   1:L PR[91] R[100]mm/sec CNT100;
   1:  PR[91,1] = PR[90,1] + -30.737;
   1:  PR[91,2] = PR[90,2] + -9.914;
   1:  PR[91,3] = PR[90,3] + 25.010;
   1:L PR[91] R[100]mm/sec CNT100;
   1:  PR[91,1] = PR[90,1] + -30.187;
   1:  PR[91,2] = PR[90,2] + -10.601;
   1:  PR[91,3] = PR[90,3] + 25.017;
   1:L PR[91] R[100]mm/sec CNT100;
   1:  PR[91,1] = PR[90,1] + -29.601;
   1:  PR[91,2] = PR[90,2] + -11.262;
   1:  PR[91,3] = PR[90,3] + 25.023;
   1:L PR[91] R[100]mm/sec CNT100;
   1:  PR[91,1] = PR[90,1] + -29.004;
   1:  PR[91,2] = PR[90,2] + -11.869;
   1:  PR[91,3] = PR[90,3] + 25.030;
   1:L PR[91] R[100]mm/sec CNT100;
   1:  PR[91,1] = PR[90,1] + -28.333;
   1:  PR[91,2] = PR[90,2] + -12.488;
   1:  PR[91,3] = PR[90,3] + 25.036;
   1:L PR[91] R[100]mm/sec CNT100;
   1:  PR[91,1] = PR[90,1] + -27.720;
   1:  PR[91,2] = PR[90,2] + -13.002;
   1:  PR[91,3] = PR[90,3] + 25.043;
   1:L PR[91] R[100]mm/sec CNT100;
   1:  PR[91,1] = PR[90,1] + -27.130;
   1:  PR[91,2] = PR[90,2] + -13.455;
   1:  PR[91,3] = PR[90,3] + 25.048;
   1:L PR[91] R[100]mm/sec CNT100;
   1:  PR[91,1] = PR[90,1] + -26.284;
   1:  PR[91,2] = PR[90,2] + -14.048;
   1:  PR[91,3] = PR[90,3] + 25.054;
   1:L PR[91] R[100]mm/sec CNT100;
   1:  PR[91,1] = PR[90,1] + -25.283;
   1:  PR[91,2] = PR[90,2] + -14.665;
   1:  PR[91,3] = PR[90,3] + 25.061;
   1:L PR[91] R[100]mm/sec CNT100;
   1:  PR[91,1] = PR[90,1] + -24.683;
   1:  PR[91,2] = PR[90,2] + -14.996;
   1:  PR[91,3] = PR[90,3] + 25.070;
   1:L PR[91] R[100]mm/sec CNT100;
   1:  PR[91,1] = PR[90,1] + -24.117;
   1:  PR[91,2] = PR[90,2] + -15.284;
   1:  PR[91,3] = PR[90,3] + 25.075;
   1:L PR[91] R[100]mm/sec CNT100;
   1:  PR[91,1] = PR[90,1] + -23.525;
   1:  PR[91,2] = PR[90,2] + -15.562;
   1:  PR[91,3] = PR[90,3] + 25.080;
   1:L PR[91] R[100]mm/sec CNT100;
   1:  PR[91,1] = PR[90,1] + -22.891;
   1:  PR[91,2] = PR[90,2] + -15.833;
   1:  PR[91,3] = PR[90,3] + 25.084;
   1:L PR[91] R[100]mm/sec CNT100;
   1:  PR[91,1] = PR[90,1] + -21.711;
   1:  PR[91,2] = PR[90,2] + -16.271;
   1:  PR[91,3] = PR[90,3] + 25.090;
   1:L PR[91] R[100]mm/sec CNT100;
   1:  PR[91,1] = PR[90,1] + -20.572;
   1:  PR[91,2] = PR[90,2] + -16.615;
   1:  PR[91,3] = PR[90,3] + 25.099;
   1:L PR[91] R[100]mm/sec CNT100;
   1:  PR[91,1] = PR[90,1] + -19.827;
   1:  PR[91,2] = PR[90,2] + -16.801;
   1:  PR[91,3] = PR[90,3] + 25.107;
   1:L PR[91] R[100]mm/sec CNT100;
   1:  PR[91,1] = PR[90,1] + -19.025;
   1:  PR[91,2] = PR[90,2] + -16.967;
   1:  PR[91,3] = PR[90,3] + 25.113;
   1:L PR[91] R[100]mm/sec CNT100;
   1:  PR[91,1] = PR[90,1] + -17.886;
   1:  PR[91,2] = PR[90,2] + -17.146;
   1:  PR[91,3] = PR[90,3] + 25.119;
   1:L PR[91] R[100]mm/sec CNT100;
   1:  PR[91,1] = PR[90,1] + -16.804;
   1:  PR[91,2] = PR[90,2] + -17.255;
   1:  PR[91,3] = PR[90,3] + 25.127;
   1:L PR[91] R[100]mm/sec CNT100;
   1:  PR[91,1] = PR[90,1] + -15.773;
   1:  PR[91,2] = PR[90,2] + -17.303;
   1:  PR[91,3] = PR[90,3] + 25.135;
   1:L PR[91] R[100]mm/sec CNT100;
   1:  PR[91,1] = PR[90,1] + -14.875;
   1:  PR[91,2] = PR[90,2] + -17.304;
   1:  PR[91,3] = PR[90,3] + 25.143;
   1:L PR[91] R[100]mm/sec CNT100;
   1:  PR[91,1] = PR[90,1] + -13.925;
   1:  PR[91,2] = PR[90,2] + -17.261;
   1:  PR[91,3] = PR[90,3] + 25.149;
   1:L PR[91] R[100]mm/sec CNT100;
   1:  PR[91,1] = PR[90,1] + -12.934;
   1:  PR[91,2] = PR[90,2] + -17.168;
   1:  PR[91,3] = PR[90,3] + 25.156;
   1:L PR[91] R[100]mm/sec CNT100;
   1:  PR[91,1] = PR[90,1] + -11.948;
   1:  PR[91,2] = PR[90,2] + -17.028;
   1:  PR[91,3] = PR[90,3] + 25.164;
   1:L PR[91] R[100]mm/sec CNT100;
   1:  PR[91,1] = PR[90,1] + -10.972;
   1:  PR[91,2] = PR[90,2] + -16.838;
   1:  PR[91,3] = PR[90,3] + 25.171;
   1:L PR[91] R[100]mm/sec CNT100;
   1:  PR[91,1] = PR[90,1] + -10.260;
   1:  PR[91,2] = PR[90,2] + -16.664;
   1:  PR[91,3] = PR[90,3] + 25.178;
   1:L PR[91] R[100]mm/sec CNT100;
   1:  PR[91,1] = PR[90,1] + -9.055;
   1:  PR[91,2] = PR[90,2] + -16.313;
   1:  PR[91,3] = PR[90,3] + 25.184;
   1:L PR[91] R[100]mm/sec CNT100;
   1:  PR[91,1] = PR[90,1] + -8.123;
   1:  PR[91,2] = PR[90,2] + -15.980;
   1:  PR[91,3] = PR[90,3] + 25.193;
   1:L PR[91] R[100]mm/sec CNT100;
   1:  PR[91,1] = PR[90,1] + -7.209;
   1:  PR[91,2] = PR[90,2] + -15.599;
   1:  PR[91,3] = PR[90,3] + 25.200;
   1:L PR[91] R[100]mm/sec CNT100;
   1:  PR[91,1] = PR[90,1] + -6.317;
   1:  PR[91,2] = PR[90,2] + -15.173;
   1:  PR[91,3] = PR[90,3] + 25.207;
   1:L PR[91] R[100]mm/sec CNT100;
   1:  PR[91,1] = PR[90,1] + -5.448;
   1:  PR[91,2] = PR[90,2] + -14.703;
   1:  PR[91,3] = PR[90,3] + 25.214;
   1:L PR[91] R[100]mm/sec CNT100;
   1:  PR[91,1] = PR[90,1] + -5.165;
   1:  PR[91,2] = PR[90,2] + -14.532;
   1:  PR[91,3] = PR[90,3] + 25.222;
   1:L PR[91] R[100]mm/sec CNT100;
   1:  PR[91,1] = PR[90,1] + -4.610;
   1:  PR[91,2] = PR[90,2] + -14.191;
   1:  PR[91,3] = PR[90,3] + 25.224;
   1:L PR[91] R[100]mm/sec CNT100;
   1:  PR[91,1] = PR[90,1] + -3.799;
   1:  PR[91,2] = PR[90,2] + -13.637;
   1:  PR[91,3] = PR[90,3] + 25.229;
   1:L PR[91] R[100]mm/sec CNT100;
   1:  PR[91,1] = PR[90,1] + -3.024;
   1:  PR[91,2] = PR[90,2] + -13.044;
   1:  PR[91,3] = PR[90,3] + 25.236;
   1:L PR[91] R[100]mm/sec CNT100;
   1:  PR[91,1] = PR[90,1] + -2.098;
   1:  PR[91,2] = PR[90,2] + -12.241;
   1:  PR[91,3] = PR[90,3] + 25.243;
   1:L PR[91] R[100]mm/sec CNT100;
   1:  PR[91,1] = PR[90,1] + -1.734;
   1:  PR[91,2] = PR[90,2] + -11.953;
   1:  PR[91,3] = PR[90,3] + 25.252;
   1:L PR[91] R[100]mm/sec CNT100;
   1:  PR[91,1] = PR[90,1] + -1.300;
   1:  PR[91,2] = PR[90,2] + -11.713;
   1:  PR[91,3] = PR[90,3] + 25.256;
   1:L PR[91] R[100]mm/sec CNT100;
   1:  PR[91,1] = PR[90,1] + -0.832;
   1:  PR[91,2] = PR[90,2] + -11.548;
   1:  PR[91,3] = PR[90,3] + 25.259;
   1:L PR[91] R[100]mm/sec CNT100;
   1:  PR[91,1] = PR[90,1] + -0.345;
   1:  PR[91,2] = PR[90,2] + -11.469;
   1:  PR[91,3] = PR[90,3] + 25.263;
   1:L PR[91] R[100]mm/sec CNT100;
   1:  PR[91,1] = PR[90,1] + 0.152;
   1:  PR[91,2] = PR[90,2] + -11.471;
   1:  PR[91,3] = PR[90,3] + 25.266;
   1:L PR[91] R[100]mm/sec CNT100;
   1:  PR[91] = PR[90];
   1:  PR[91,1] = PR[90,1] + 0.746;
   1:  PR[91,2] = PR[90,2] + -12.225;
   1:  PR[91,3] = PR[90,3] + 26.600;
   1:L PR[91] R[100]mm/sec CNT100;
   1:  PR[91,1] = PR[90,1] + 1.211;
   1:  PR[91,2] = PR[90,2] + -12.418;
   1:  PR[91,3] = PR[90,3] + 25.274;
   1:L PR[91] R[100]mm/sec CNT100;
   1:  PR[91,1] = PR[90,1] + 1.632;
   1:  PR[91,2] = PR[90,2] + -12.682;
   1:  PR[91,3] = PR[90,3] + 25.277;
   1:L PR[91] R[100]mm/sec CNT100;
   1:  PR[91,1] = PR[90,1] + 2.218;
   1:  PR[91,2] = PR[90,2] + -13.167;
   1:  PR[91,3] = PR[90,3] + 25.281;
   1:L PR[91] R[100]mm/sec CNT100;
   1:  PR[91,1] = PR[90,1] + 3.031;
   1:  PR[91,2] = PR[90,2] + -13.784;
   1:  PR[91,3] = PR[90,3] + 25.287;
   1:L PR[91] R[100]mm/sec CNT100;
   1:  PR[91,1] = PR[90,1] + 3.666;
   1:  PR[91,2] = PR[90,2] + -14.220;
   1:  PR[91,3] = PR[90,3] + 25.294;
   1:L PR[91] R[100]mm/sec CNT100;
   1:  PR[91,1] = PR[90,1] + 4.499;
   1:  PR[91,2] = PR[90,2] + -14.736;
   1:  PR[91,3] = PR[90,3] + 25.300;
   1:L PR[91] R[100]mm/sec CNT100;
   1:  PR[91,1] = PR[90,1] + 5.359;
   1:  PR[91,2] = PR[90,2] + -15.209;
   1:  PR[91,3] = PR[90,3] + 25.307;
   1:L PR[91] R[100]mm/sec CNT100;
   1:  PR[91,1] = PR[90,1] + 6.243;
   1:  PR[91,2] = PR[90,2] + -15.639;
   1:  PR[91,3] = PR[90,3] + 25.314;
   1:L PR[91] R[100]mm/sec CNT100;
   1:  PR[91,1] = PR[90,1] + 7.150;
   1:  PR[91,2] = PR[90,2] + -16.025;
   1:  PR[91,3] = PR[90,3] + 25.322;
   1:L PR[91] R[100]mm/sec CNT100;
   1:  PR[91,1] = PR[90,1] + 8.081;
   1:  PR[91,2] = PR[90,2] + -16.368;
   1:  PR[91,3] = PR[90,3] + 25.329;
   1:L PR[91] R[100]mm/sec CNT100;
   1:  PR[91,1] = PR[90,1] + 9.032;
   1:  PR[91,2] = PR[90,2] + -16.664;
   1:  PR[91,3] = PR[90,3] + 25.336;
   1:L PR[91] R[100]mm/sec CNT100;
   1:  PR[91,1] = PR[90,1] + 10.000;
   1:  PR[91,2] = PR[90,2] + -16.914;
   1:  PR[91,3] = PR[90,3] + 25.344;
   1:L PR[91] R[100]mm/sec CNT100;
   1:  PR[91,1] = PR[90,1] + 10.985;
   1:  PR[91,2] = PR[90,2] + -17.116;
   1:  PR[91,3] = PR[90,3] + 25.351;
   1:L PR[91] R[100]mm/sec CNT100;
   1:  PR[91,1] = PR[90,1] + 11.982;
   1:  PR[91,2] = PR[90,2] + -17.268;
   1:  PR[91,3] = PR[90,3] + 25.359;
   1:L PR[91] R[100]mm/sec CNT100;
   1:  PR[91,1] = PR[90,1] + 12.990;
   1:  PR[91,2] = PR[90,2] + -17.370;
   1:  PR[91,3] = PR[90,3] + 25.366;
   1:L PR[91] R[100]mm/sec CNT100;
   1:  PR[91,1] = PR[90,1] + 14.005;
   1:  PR[91,2] = PR[90,2] + -17.420;
   1:  PR[91,3] = PR[90,3] + 25.374;
   1:L PR[91] R[100]mm/sec CNT100;
   1:  PR[91,1] = PR[90,1] + 15.024;
   1:  PR[91,3] = PR[90,3] + 25.381;
   1:L PR[91] R[100]mm/sec CNT100;
   1:  PR[91,1] = PR[90,1] + 16.046;
   1:  PR[91,2] = PR[90,2] + -17.368;
   1:  PR[91,3] = PR[90,3] + 25.389;
   1:L PR[91] R[100]mm/sec CNT100;
   1:  PR[91,1] = PR[90,1] + 17.066;
   1:  PR[91,2] = PR[90,2] + -17.265;
   1:  PR[91,3] = PR[90,3] + 25.396;
   1:L PR[91] R[100]mm/sec CNT100;
   1:  PR[91,1] = PR[90,1] + 18.089;
   1:  PR[91,2] = PR[90,2] + -17.108;
   1:  PR[91,3] = PR[90,3] + 25.404;
   1:L PR[91] R[100]mm/sec CNT100;
   1:  PR[91,1] = PR[90,1] + 19.054;
   1:  PR[91,2] = PR[90,2] + -16.911;
   1:  PR[91,3] = PR[90,3] + 25.411;
   1:L PR[91] R[100]mm/sec CNT100;
   1:  PR[91,1] = PR[90,1] + 19.959;
   1:  PR[91,2] = PR[90,2] + -16.682;
   1:  PR[91,3] = PR[90,3] + 25.419;
   1:L PR[91] R[100]mm/sec CNT100;
   1:  PR[91,1] = PR[90,1] + 20.950;
   1:  PR[91,2] = PR[90,2] + -16.379;
   1:  PR[91,3] = PR[90,3] + 25.426;
   1:L PR[91] R[100]mm/sec CNT100;
   1:  PR[91,1] = PR[90,1] + 21.772;
   1:  PR[91,2] = PR[90,2] + -16.084;
   1:  PR[91,3] = PR[90,3] + 25.433;
   1:L PR[91] R[100]mm/sec CNT100;
   1:  PR[91,1] = PR[90,1] + 22.540;
   1:  PR[91,2] = PR[90,2] + -15.769;
   1:  PR[91,3] = PR[90,3] + 25.440;
   1:L PR[91] R[100]mm/sec CNT100;
   1:  PR[91,1] = PR[90,1] + 23.029;
   1:  PR[91,2] = PR[90,2] + -15.550;
   1:  PR[91,3] = PR[90,3] + 25.446;
   1:L PR[91] R[100]mm/sec CNT100;
   1:  PR[91,1] = PR[90,1] + 23.799;
   1:  PR[91,2] = PR[90,2] + -15.175;
   1:  PR[91,3] = PR[90,3] + 25.450;
   1:L PR[91] R[100]mm/sec CNT100;
   1:  PR[91,1] = PR[90,1] + 24.506;
   1:  PR[91,2] = PR[90,2] + -14.792;
   1:  PR[91,3] = PR[90,3] + 25.456;
   1:L PR[91] R[100]mm/sec CNT100;
   1:  PR[91,1] = PR[90,1] + 25.155;
   1:  PR[91,2] = PR[90,2] + -14.404;
   1:  PR[91,3] = PR[90,3] + 25.462;
   1:L PR[91] R[100]mm/sec CNT100;
   1:  PR[91,1] = PR[90,1] + 26.123;
   1:  PR[91,2] = PR[90,2] + -13.760;
   1:  PR[91,3] = PR[90,3] + 25.468;
   1:L PR[91] R[100]mm/sec CNT100;
   1:  PR[91,1] = PR[90,1] + 27.087;
   1:  PR[91,2] = PR[90,2] + -13.027;
   1:  PR[91,3] = PR[90,3] + 25.476;
   1:L PR[91] R[100]mm/sec CNT100;
   1:  PR[91,1] = PR[90,1] + 27.605;
   1:  PR[91,2] = PR[90,2] + -12.590;
   1:  PR[91,3] = PR[90,3] + 25.485;
   1:L PR[91] R[100]mm/sec CNT100;
   1:  PR[91,1] = PR[90,1] + 28.084;
   1:  PR[91,2] = PR[90,2] + -12.156;
   1:  PR[91,3] = PR[90,3] + 25.490;
   1:L PR[91] R[100]mm/sec CNT100;
   1:  PR[91,1] = PR[90,1] + 28.505;
   1:  PR[91,2] = PR[90,2] + -11.747;
   1:  PR[91,3] = PR[90,3] + 25.495;
   1:L PR[91] R[100]mm/sec CNT100;
   1:  PR[91,1] = PR[90,1] + 28.938;
   1:  PR[91,2] = PR[90,2] + -11.297;
   1:  PR[91,3] = PR[90,3] + 25.499;
   1:L PR[91] R[100]mm/sec CNT100;
   1:  PR[91,1] = PR[90,1] + 29.365;
   1:  PR[91,2] = PR[90,2] + -10.820;
   1:  PR[91,3] = PR[90,3] + 25.504;
   1:L PR[91] R[100]mm/sec CNT100;
   1:  PR[91,1] = PR[90,1] + 30.117;
   1:  PR[91,2] = PR[90,2] + -9.888;
   1:  PR[91,3] = PR[90,3] + 25.509;
   1:L PR[91] R[100]mm/sec CNT100;
   1:  PR[91,1] = PR[90,1] + 30.525;
   1:  PR[91,2] = PR[90,2] + -9.323;
   1:  PR[91,3] = PR[90,3] + 25.518;
   1:L PR[91] R[100]mm/sec CNT100;
   1:  PR[91,1] = PR[90,1] + 31.132;
   1:  PR[91,2] = PR[90,2] + -8.387;
   1:  PR[91,3] = PR[90,3] + 25.523;
   1:L PR[91] R[100]mm/sec CNT100;
   1:  PR[91,1] = PR[90,1] + 31.502;
   1:  PR[91,2] = PR[90,2] + -7.751;
   1:  PR[91,3] = PR[90,3] + 25.531;
   1:L PR[91] R[100]mm/sec CNT100;
   1:  PR[91,1] = PR[90,1] + 31.859;
   1:  PR[91,2] = PR[90,2] + -7.073;
   1:  PR[91,3] = PR[90,3] + 25.536;
   1:L PR[91] R[100]mm/sec CNT100;
   1:  PR[91,1] = PR[90,1] + 32.291;
   1:  PR[91,2] = PR[90,2] + -6.150;
   1:  PR[91,3] = PR[90,3] + 25.542;
   1:L PR[91] R[100]mm/sec CNT100;
   1:  PR[91,1] = PR[90,1] + 32.582;
   1:  PR[91,2] = PR[90,2] + -5.440;
   1:  PR[91,3] = PR[90,3] + 25.550;
   1:L PR[91] R[100]mm/sec CNT100;
   1:  PR[91,1] = PR[90,1] + 32.844;
   1:  PR[91,2] = PR[90,2] + -4.705;
   1:  PR[91,3] = PR[90,3] + 25.555;
   1:L PR[91] R[100]mm/sec CNT100;
   1:  PR[91,1] = PR[90,1] + 33.106;
   1:  PR[91,2] = PR[90,2] + -3.830;
   1:  PR[91,3] = PR[90,3] + 25.561;
   1:L PR[91] R[100]mm/sec CNT100;
   1:  PR[91,1] = PR[90,1] + 33.290;
   1:  PR[91,2] = PR[90,2] + -3.066;
   1:  PR[91,3] = PR[90,3] + 25.568;
   1:L PR[91] R[100]mm/sec CNT100;
   1:  PR[91,1] = PR[90,1] + 33.451;
   1:  PR[91,2] = PR[90,2] + -2.189;
   1:  PR[91,3] = PR[90,3] + 25.574;
   1:L PR[91] R[100]mm/sec CNT100;
   1:  PR[91,1] = PR[90,1] + 33.555;
   1:  PR[91,2] = PR[90,2] + -1.373;
   1:  PR[91,3] = PR[90,3] + 25.580;
   1:L PR[91] R[100]mm/sec CNT100;
   1:  PR[91,1] = PR[90,1] + 33.624;
   1:  PR[91,2] = PR[90,2] + -0.455;
   1:  PR[91,3] = PR[90,3] + 25.586;
   1:L PR[91] R[100]mm/sec CNT100;
   1:  PR[91,1] = PR[90,1] + 33.645;
   1:  PR[91,2] = PR[90,2] + 0.427;
   1:  PR[91,3] = PR[90,3] + 25.593;
   1:L PR[91] R[100]mm/sec CNT100;
   1:  PR[91,1] = PR[90,1] + 33.620;
   1:  PR[91,2] = PR[90,2] + 1.378;
   1:  PR[91,3] = PR[90,3] + 25.600;
   1:L PR[91] R[100]mm/sec CNT100;
   1:  PR[91,1] = PR[90,1] + 33.555;
   1:  PR[91,2] = PR[90,2] + 2.228;
   1:  PR[91,3] = PR[90,3] + 25.607;
   1:L PR[91] R[100]mm/sec CNT100;
   1:  PR[91,1] = PR[90,1] + 33.451;
   1:  PR[91,2] = PR[90,2] + 3.044;
   1:  PR[91,3] = PR[90,3] + 25.613;
   1:L PR[91] R[100]mm/sec CNT100;
   1:  PR[91,1] = PR[90,1] + 33.290;
   1:  PR[91,2] = PR[90,2] + 3.921;
   1:  PR[91,3] = PR[90,3] + 25.619;
   1:L PR[91] R[100]mm/sec CNT100;
   1:  PR[91,1] = PR[90,1] + 33.106;
   1:  PR[91,2] = PR[90,2] + 4.686;
   1:  PR[91,3] = PR[90,3] + 25.626;
   1:L PR[91] R[100]mm/sec CNT100;
   1:  PR[91,1] = PR[90,1] + 32.888;
   1:  PR[91,2] = PR[90,2] + 5.423;
   1:  PR[91,3] = PR[90,3] + 25.632;
   1:L PR[91] R[100]mm/sec CNT100;
   1:  PR[91,1] = PR[90,1] + 32.581;
   1:  PR[91,2] = PR[90,2] + 6.296;
   1:  PR[91,3] = PR[90,3] + 25.637;
   1:L PR[91] R[100]mm/sec CNT100;
   1:  PR[91,1] = PR[90,1] + 32.291;
   1:  PR[91,2] = PR[90,2] + 7.006;
   1:  PR[91,3] = PR[90,3] + 25.644;
   1:L PR[91] R[100]mm/sec CNT100;
   1:  PR[91,1] = PR[90,1] + 31.975;
   1:  PR[91,2] = PR[90,2] + 7.691;
   1:  PR[91,3] = PR[90,3] + 25.650;
   1:L PR[91] R[100]mm/sec CNT100;
   1:  PR[91,1] = PR[90,1] + 31.501;
   1:  PR[91,2] = PR[90,2] + 8.608;
   1:  PR[91,3] = PR[90,3] + 25.655;
   1:L PR[91] R[100]mm/sec CNT100;
   1:  PR[91,1] = PR[90,1] + 31.131;
   1:  PR[91,2] = PR[90,2] + 9.244;
   1:  PR[91,3] = PR[90,3] + 25.663;
   1:L PR[91] R[100]mm/sec CNT100;
   1:  PR[91,1] = PR[90,1] + 30.753;
   1:  PR[91,2] = PR[90,2] + 9.838;
   1:  PR[91,3] = PR[90,3] + 25.668;
   1:L PR[91] R[100]mm/sec CNT100;
   1:  PR[91,1] = PR[90,1] + 30.111;
   1:  PR[91,2] = PR[90,2] + 10.750;
   1:  PR[91,3] = PR[90,3] + 25.674;
   1:L PR[91] R[100]mm/sec CNT100;
   1:  PR[91,1] = PR[90,1] + 29.810;
   1:  PR[91,2] = PR[90,2] + 11.137;
   1:  PR[91,3] = PR[90,3] + 25.682;
   1:L PR[91] R[100]mm/sec CNT100;
   1:  PR[91,1] = PR[90,1] + 29.368;
   1:  PR[91,2] = PR[90,2] + 11.672;
   1:  PR[91,3] = PR[90,3] + 25.686;
   1:L PR[91] R[100]mm/sec CNT100;
   1:  PR[91,1] = PR[90,1] + 28.938;
   1:  PR[91,2] = PR[90,2] + 12.152;
   1:  PR[91,3] = PR[90,3] + 25.691;
   1:L PR[91] R[100]mm/sec CNT100;
   1:  PR[91,1] = PR[90,1] + 28.505;
   1:  PR[91,2] = PR[90,2] + 12.602;
   1:  PR[91,3] = PR[90,3] + 25.695;
   1:L PR[91] R[100]mm/sec CNT100;
   1:  PR[91,1] = PR[90,1] + 28.084;
   1:  PR[91,2] = PR[90,2] + 13.011;
   1:  PR[91,3] = PR[90,3] + 25.700;
   1:L PR[91] R[100]mm/sec CNT100;
   1:  PR[91,1] = PR[90,1] + 27.605;
   1:  PR[91,2] = PR[90,2] + 13.446;
   1:  PR[91,3] = PR[90,3] + 25.704;
   1:L PR[91] R[100]mm/sec CNT100;
   1:  PR[91,1] = PR[90,1] + 27.087;
   1:  PR[91,2] = PR[90,2] + 13.882;
   1:  PR[91,3] = PR[90,3] + 25.709;
   1:L PR[91] R[100]mm/sec CNT100;
   1:  PR[91,1] = PR[90,1] + 26.123;
   1:  PR[91,2] = PR[90,2] + 14.615;
   1:  PR[91,3] = PR[90,3] + 25.714;
   1:L PR[91] R[100]mm/sec CNT100;
   1:  PR[91,1] = PR[90,1] + 25.155;
   1:  PR[91,2] = PR[90,2] + 15.259;
   1:  PR[91,3] = PR[90,3] + 25.723;
   1:L PR[91] R[100]mm/sec CNT100;
   1:  PR[91,1] = PR[90,1] + 24.508;
   1:  PR[91,2] = PR[90,2] + 15.646;
   1:  PR[91,3] = PR[90,3] + 25.732;
   1:L PR[91] R[100]mm/sec CNT100;
   1:  PR[91,1] = PR[90,1] + 23.509;
   1:  PR[91,2] = PR[90,2] + 16.177;
   1:  PR[91,3] = PR[90,3] + 25.737;
   1:L PR[91] R[100]mm/sec CNT100;
   1:  PR[91,1] = PR[90,1] + 22.773;
   1:  PR[91,2] = PR[90,2] + 16.525;
   1:  PR[91,3] = PR[90,3] + 25.746;
   1:L PR[91] R[100]mm/sec CNT100;
   1:  PR[91,1] = PR[90,1] + 21.975;
   1:  PR[91,2] = PR[90,2] + 16.860;
   1:  PR[91,3] = PR[90,3] + 25.752;
   1:L PR[91] R[100]mm/sec CNT100;
   1:  PR[91,1] = PR[90,1] + 20.948;
   1:  PR[91,2] = PR[90,2] + 17.235;
   1:  PR[91,3] = PR[90,3] + 25.758;
   1:L PR[91] R[100]mm/sec CNT100;
   1:  PR[91,1] = PR[90,1] + 19.958;
   1:  PR[91,2] = PR[90,2] + 17.537;
   1:  PR[91,3] = PR[90,3] + 25.766;
   1:L PR[91] R[100]mm/sec CNT100;
   1:  PR[91,1] = PR[90,1] + 19.054;
   1:  PR[91,2] = PR[90,2] + 17.767;
   1:  PR[91,3] = PR[90,3] + 25.774;
   1:L PR[91] R[100]mm/sec CNT100;
   1:  PR[91,1] = PR[90,1] + 18.081;
   1:  PR[91,2] = PR[90,2] + 17.964;
   1:  PR[91,3] = PR[90,3] + 25.781;
   1:L PR[91] R[100]mm/sec CNT100;
   1:  PR[91,1] = PR[90,1] + 17.065;
   1:  PR[91,2] = PR[90,2] + 18.120;
   1:  PR[91,3] = PR[90,3] + 25.788;
   1:L PR[91] R[100]mm/sec CNT100;
   1:  PR[91,1] = PR[90,1] + 16.045;
   1:  PR[91,2] = PR[90,2] + 18.223;
   1:  PR[91,3] = PR[90,3] + 25.796;
   1:L PR[91] R[100]mm/sec CNT100;
   1:  PR[91,1] = PR[90,1] + 15.024;
   1:  PR[91,2] = PR[90,2] + 18.275;
   1:  PR[91,3] = PR[90,3] + 25.803;
   1:L PR[91] R[100]mm/sec CNT100;
   1:  PR[91,1] = PR[90,1] + 14.002;
   1:  PR[91,2] = PR[90,2] + 18.276;
   1:  PR[91,3] = PR[90,3] + 25.811;
   1:L PR[91] R[100]mm/sec CNT100;
   1:  PR[91,1] = PR[90,1] + 13.394;
   1:  PR[91,2] = PR[90,2] + 18.250;
   1:  PR[91,3] = PR[90,3] + 25.818;
   1:L PR[91] R[100]mm/sec CNT100;
   1:  PR[91,1] = PR[90,1] + 12.993;
   1:  PR[91,2] = PR[90,2] + 18.225;
   1:  PR[91,3] = PR[90,3] + 25.823;
   1:L PR[91] R[100]mm/sec CNT100;
   1:  PR[91,1] = PR[90,1] + 11.982;
   1:  PR[91,2] = PR[90,2] + 18.123;
   1:  PR[91,3] = PR[90,3] + 25.826;
   1:L PR[91] R[100]mm/sec CNT100;
   1:  PR[91,1] = PR[90,1] + 10.982;
   1:  PR[91,2] = PR[90,2] + 17.970;
   1:  PR[91,3] = PR[90,3] + 25.833;
   1:L PR[91] R[100]mm/sec CNT100;
   1:  PR[91,1] = PR[90,1] + 10.618;
   1:  PR[91,2] = PR[90,2] + 17.900;
   1:  PR[91,3] = PR[90,3] + 25.841;
   1:L PR[91] R[100]mm/sec CNT100;
   1:  PR[91,1] = PR[90,1] + 10.003;
   1:  PR[91,2] = PR[90,2] + 17.770;
   1:  PR[91,3] = PR[90,3] + 25.844;
   1:L PR[91] R[100]mm/sec CNT100;
   1:  PR[91,1] = PR[90,1] + 9.032;
   1:  PR[91,2] = PR[90,2] + 17.520;
   1:  PR[91,3] = PR[90,3] + 25.848;
   1:L PR[91] R[100]mm/sec CNT100;
   1:  PR[91,1] = PR[90,1] + 8.081;
   1:  PR[91,2] = PR[90,2] + 17.223;
   1:  PR[91,3] = PR[90,3] + 25.856;
   1:L PR[91] R[100]mm/sec CNT100;
   1:  PR[91,1] = PR[90,1] + 7.151;
   1:  PR[91,2] = PR[90,2] + 16.881;
   1:  PR[91,3] = PR[90,3] + 25.863;
   1:L PR[91] R[100]mm/sec CNT100;
   1:  PR[91,1] = PR[90,1] + 6.243;
   1:  PR[91,2] = PR[90,2] + 16.494;
   1:  PR[91,3] = PR[90,3] + 25.870;
   1:L PR[91] R[100]mm/sec CNT100;
   1:  PR[91,1] = PR[90,1] + 5.359;
   1:  PR[91,2] = PR[90,2] + 16.064;
   1:  PR[91,3] = PR[90,3] + 25.878;
   1:L PR[91] R[100]mm/sec CNT100;
   1:  PR[91,1] = PR[90,1] + 4.499;
   1:  PR[91,2] = PR[90,2] + 15.591;
   1:  PR[91,3] = PR[90,3] + 25.885;
   1:L PR[91] R[100]mm/sec CNT100;
   1:  PR[91,1] = PR[90,1] + 3.794;
   1:  PR[91,2] = PR[90,2] + 15.157;
   1:  PR[91,3] = PR[90,3] + 25.892;
   1:L PR[91] R[100]mm/sec CNT100;
   1:  PR[91,1] = PR[90,1] + 2.863;
   1:  PR[91,2] = PR[90,2] + 14.519;
   1:  PR[91,3] = PR[90,3] + 25.898;
   1:L PR[91] R[100]mm/sec CNT100;
   1:  PR[91,1] = PR[90,1] + 2.220;
   1:  PR[91,2] = PR[90,2] + 14.024;
   1:  PR[91,3] = PR[90,3] + 25.907;
   1:L PR[91] R[100]mm/sec CNT100;
   1:  PR[91,1] = PR[90,1] + 1.632;
   1:  PR[91,2] = PR[90,2] + 13.537;
   1:  PR[91,3] = PR[90,3] + 25.913;
   1:L PR[91] R[100]mm/sec CNT100;
   1:  PR[91,1] = PR[90,1] + 1.211;
   1:  PR[91,2] = PR[90,2] + 13.274;
   1:  PR[91,3] = PR[90,3] + 25.918;
   1:L PR[91] R[100]mm/sec CNT100;
   1:  PR[91,1] = PR[90,1] + 0.746;
   1:  PR[91,2] = PR[90,2] + 13.080;
   1:  PR[91,3] = PR[90,3] + 25.922;
   1:L PR[91] R[100]mm/sec CNT100;
   1:  PR[91,1] = PR[90,1] + 0.256;
   1:  PR[91,2] = PR[90,2] + 12.971;
   1:  PR[91,3] = PR[90,3] + 25.926;
   1:L PR[91] R[100]mm/sec CNT100;
   1:  PR[91,1] = PR[90,1] + -0.239;
   1:  PR[91,2] = PR[90,2] + 12.949;
   1:  PR[91,3] = PR[90,3] + 25.929;
   1:L PR[91] R[100]mm/sec CNT100;
   1:  PR[91,1] = PR[90,1] + -0.723;
   1:  PR[91,2] = PR[90,2] + 13.011;
   1:  PR[91,3] = PR[90,3] + 25.933;
   1:L PR[91] R[100]mm/sec CNT100;
   1:  PR[91,1] = PR[90,1] + -0.967;
   1:  PR[91,2] = PR[90,2] + 13.081;
   1:  PR[91,3] = PR[90,3] + 25.937;
   1:L PR[91] R[100]mm/sec CNT100;
   1:  PR[91,1] = PR[90,1] + -1.206;
   1:  PR[91,2] = PR[90,2] + 13.159;
   1:  PR[91,3] = PR[90,3] + 25.939;
   1:L PR[91] R[100]mm/sec CNT100;
   1:  PR[91,1] = PR[90,1] + -1.645;
   1:  PR[91,2] = PR[90,2] + 13.379;
   1:  PR[91,3] = PR[90,3] + 25.940;
   1:L PR[91] R[100]mm/sec CNT100;
   1:  PR[91,1] = PR[90,1] + -2.022;
   1:  PR[91,2] = PR[90,2] + 13.658;
   1:  PR[91,3] = PR[90,3] + 25.944;
   1:L PR[91] R[100]mm/sec CNT100;
   1:  PR[91,1] = PR[90,1] + -2.509;
   1:  PR[91,2] = PR[90,2] + 14.062;
   1:  PR[91,3] = PR[90,3] + 25.948;
   1:L PR[91] R[100]mm/sec CNT100;
   1:  PR[91,1] = PR[90,1] + -3.128;
   1:  PR[91,2] = PR[90,2] + 14.535;
   1:  PR[91,3] = PR[90,3] + 25.952;
   1:L PR[91] R[100]mm/sec CNT100;
   1:  PR[91,1] = PR[90,1] + -3.950;
   1:  PR[91,2] = PR[90,2] + 15.102;
   1:  PR[91,3] = PR[90,3] + 25.958;
   1:L PR[91] R[100]mm/sec CNT100;
   1:  PR[91,1] = PR[90,1] + -4.805;
   1:  PR[91,2] = PR[90,2] + 15.627;
   1:  PR[91,3] = PR[90,3] + 25.965;
   1:L PR[91] R[100]mm/sec CNT100;
   1:  PR[91,1] = PR[90,1] + -5.713;
   1:  PR[91,2] = PR[90,2] + 16.121;
   1:  PR[91,3] = PR[90,3] + 25.973;
   1:L PR[91] R[100]mm/sec CNT100;
   1:  PR[91,1] = PR[90,1] + -6.594;
   1:  PR[91,2] = PR[90,2] + 16.545;
   1:  PR[91,3] = PR[90,3] + 25.980;
   1:L PR[91] R[100]mm/sec CNT100;
   1:  PR[91,1] = PR[90,1] + -7.514;
   1:  PR[91,2] = PR[90,2] + 16.931;
   1:  PR[91,3] = PR[90,3] + 25.988;
   1:L PR[91] R[100]mm/sec CNT100;
   1:  PR[91,1] = PR[90,1] + -8.452;
   1:  PR[91,2] = PR[90,2] + 17.270;
   1:  PR[91,3] = PR[90,3] + 25.995;
   1:L PR[91] R[100]mm/sec CNT100;
   1:  PR[91,1] = PR[90,1] + -9.408;
   1:  PR[91,2] = PR[90,2] + 17.561;
   1:  PR[91,3] = PR[90,3] + 26.002;
   1:L PR[91] R[100]mm/sec CNT100;
   1:  PR[91,1] = PR[90,1] + -10.378;
   1:  PR[91,2] = PR[90,2] + 17.803;
   1:  PR[91,3] = PR[90,3] + 26.010;
   1:L PR[91] R[100]mm/sec CNT100;
   1:  PR[91,1] = PR[90,1] + -11.359;
   1:  PR[91,2] = PR[90,2] + 17.996;
   1:  PR[91,3] = PR[90,3] + 26.017;
   1:L PR[91] R[100]mm/sec CNT100;
   1:  PR[91,1] = PR[90,1] + -12.350;
   1:  PR[91,2] = PR[90,2] + 18.140;
   1:  PR[91,3] = PR[90,3] + 26.025;
   1:L PR[91] R[100]mm/sec CNT100;
   1:  PR[91,1] = PR[90,1] + -13.346;
   1:  PR[91,2] = PR[90,2] + 18.234;
   1:  PR[91,3] = PR[90,3] + 26.032;
   1:L PR[91] R[100]mm/sec CNT100;
   1:  PR[91,1] = PR[90,1] + -14.345;
   1:  PR[91,2] = PR[90,2] + 18.278;
   1:  PR[91,3] = PR[90,3] + 26.039;
   1:L PR[91] R[100]mm/sec CNT100;
   1:  PR[91,1] = PR[90,1] + -15.344;
   1:  PR[91,2] = PR[90,2] + 18.274;
   1:  PR[91,3] = PR[90,3] + 26.047;
   1:L PR[91] R[100]mm/sec CNT100;
   1:  PR[91,1] = PR[90,1] + -16.341;
   1:  PR[91,2] = PR[90,2] + 18.219;
   1:  PR[91,3] = PR[90,3] + 26.054;
   1:L PR[91] R[100]mm/sec CNT100;
   1:  PR[91,1] = PR[90,1] + -17.331;
   1:  PR[91,2] = PR[90,2] + 18.116;
   1:  PR[91,3] = PR[90,3] + 26.062;
   1:L PR[91] R[100]mm/sec CNT100;
   1:  PR[91,1] = PR[90,1] + -18.323;
   1:  PR[91,2] = PR[90,2] + 17.963;
   1:  PR[91,3] = PR[90,3] + 26.069;
   1:L PR[91] R[100]mm/sec CNT100;
   1:  PR[91,1] = PR[90,1] + -19.288;
   1:  PR[91,2] = PR[90,2] + 17.768;
   1:  PR[91,3] = PR[90,3] + 26.076;
   1:L PR[91] R[100]mm/sec CNT100;
   1:  PR[91,1] = PR[90,1] + -20.196;
   1:  PR[91,2] = PR[90,2] + 17.539;
   1:  PR[91,3] = PR[90,3] + 26.084;
   1:L PR[91] R[100]mm/sec CNT100;
   1:  PR[91,1] = PR[90,1] + -21.189;
   1:  PR[91,2] = PR[90,2] + 17.236;
   1:  PR[91,3] = PR[90,3] + 26.091;
   1:L PR[91] R[100]mm/sec CNT100;
   1:  PR[91,1] = PR[90,1] + -22.012;
   1:  PR[91,2] = PR[90,2] + 16.940;
   1:  PR[91,3] = PR[90,3] + 26.098;
   1:L PR[91] R[100]mm/sec CNT100;
   1:  PR[91,1] = PR[90,1] + -23.016;
   1:  PR[91,2] = PR[90,2] + 16.523;
   1:  PR[91,3] = PR[90,3] + 26.105;
   1:L PR[91] R[100]mm/sec CNT100;
   1:  PR[91,1] = PR[90,1] + -23.753;
   1:  PR[91,2] = PR[90,2] + 16.174;
   1:  PR[91,3] = PR[90,3] + 26.113;
   1:L PR[91] R[100]mm/sec CNT100;
   1:  PR[91,1] = PR[90,1] + -24.756;
   1:  PR[91,2] = PR[90,2] + 15.638;
   1:  PR[91,3] = PR[90,3] + 26.119;
   1:L PR[91] R[100]mm/sec CNT100;
   1:  PR[91,1] = PR[90,1] + -25.406;
   1:  PR[91,2] = PR[90,2] + 15.249;
   1:  PR[91,3] = PR[90,3] + 26.127;
   1:L PR[91] R[100]mm/sec CNT100;
   1:  PR[91,1] = PR[90,1] + -26.386;
   1:  PR[91,2] = PR[90,2] + 14.594;
   1:  PR[91,3] = PR[90,3] + 26.133;
   1:L PR[91] R[100]mm/sec CNT100;
   1:  PR[91,1] = PR[90,1] + -26.948;
   1:  PR[91,2] = PR[90,2] + 14.178;
   1:  PR[91,3] = PR[90,3] + 26.142;
   1:L PR[91] R[100]mm/sec CNT100;
   1:  PR[91,1] = PR[90,1] + -27.884;
   1:  PR[91,2] = PR[90,2] + 13.408;
   1:  PR[91,3] = PR[90,3] + 26.147;
   1:L PR[91] R[100]mm/sec CNT100;
   1:  PR[91,1] = PR[90,1] + -28.363;
   1:  PR[91,2] = PR[90,2] + 12.972;
   1:  PR[91,3] = PR[90,3] + 26.156;
   1:L PR[91] R[100]mm/sec CNT100;
   1:  PR[91,1] = PR[90,1] + -28.804;
   1:  PR[91,2] = PR[90,2] + 12.542;
   1:  PR[91,3] = PR[90,3] + 26.160;
   1:L PR[91] R[100]mm/sec CNT100;
   1:  PR[91,1] = PR[90,1] + -29.218;
   1:  PR[91,2] = PR[90,2] + 12.111;
   1:  PR[91,3] = PR[90,3] + 26.165;
   1:L PR[91] R[100]mm/sec CNT100;
   1:  PR[91,1] = PR[90,1] + -29.640;
   1:  PR[91,2] = PR[90,2] + 11.639;
   1:  PR[91,3] = PR[90,3] + 26.169;
   1:L PR[91] R[100]mm/sec CNT100;
   1:  PR[91,1] = PR[90,1] + -30.379;
   1:  PR[91,2] = PR[90,2] + 10.721;
   1:  PR[91,3] = PR[90,3] + 26.174;
   1:L PR[91] R[100]mm/sec CNT100;
   1:  PR[91,1] = PR[90,1] + -30.782;
   1:  PR[91,2] = PR[90,2] + 10.162;
   1:  PR[91,3] = PR[90,3] + 26.183;
   1:L PR[91] R[100]mm/sec CNT100;
   1:  PR[91,1] = PR[90,1] + -31.185;
   1:  PR[91,2] = PR[90,2] + 9.551;
   1:  PR[91,3] = PR[90,3] + 26.188;
   1:L PR[91] R[100]mm/sec CNT100;
   1:  PR[91,1] = PR[90,1] + -31.747;
   1:  PR[91,2] = PR[90,2] + 8.601;
   1:  PR[91,3] = PR[90,3] + 26.193;
   1:L PR[91] R[100]mm/sec CNT100;
   1:  PR[91,1] = PR[90,1] + -32.101;
   1:  PR[91,2] = PR[90,2] + 7.923;
   1:  PR[91,3] = PR[90,3] + 26.202;
   1:L PR[91] R[100]mm/sec CNT100;
   1:  PR[91,1] = PR[90,1] + -32.533;
   1:  PR[91,2] = PR[90,2] + 6.990;
   1:  PR[91,3] = PR[90,3] + 26.207;
   1:L PR[91] R[100]mm/sec CNT100;
   1:  PR[91,1] = PR[90,1] + -32.824;
   1:  PR[91,2] = PR[90,2] + 6.273;
   1:  PR[91,3] = PR[90,3] + 26.215;
   1:L PR[91] R[100]mm/sec CNT100;
   1:  PR[91,1] = PR[90,1] + -33.086;
   1:  PR[91,2] = PR[90,2] + 5.533;
   1:  PR[91,3] = PR[90,3] + 26.221;
   1:L PR[91] R[100]mm/sec CNT100;
   1:  PR[91,1] = PR[90,1] + -33.315;
   1:  PR[91,2] = PR[90,2] + 4.772;
   1:  PR[91,3] = PR[90,3] + 26.226;
   1:L PR[91] R[100]mm/sec CNT100;
   1:  PR[91,1] = PR[90,1] + -33.531;
   1:  PR[91,2] = PR[90,2] + 3.892;
   1:  PR[91,3] = PR[90,3] + 26.232;
   1:L PR[91] R[100]mm/sec CNT100;
   1:  PR[91,1] = PR[90,1] + -33.691;
   1:  PR[91,2] = PR[90,2] + 3.023;
   1:  PR[91,3] = PR[90,3] + 26.239;
   1:L PR[91] R[100]mm/sec CNT100;
   1:  PR[91,1] = PR[90,1] + -33.795;
   1:  PR[91,2] = PR[90,2] + 2.215;
   1:  PR[91,3] = PR[90,3] + 26.245;
   1:L PR[91] R[100]mm/sec CNT100;
   1:  PR[91,1] = PR[90,1] + -33.859;
   1:  PR[91,2] = PR[90,2] + 1.371;
   1:  PR[91,3] = PR[90,3] + 26.251;
   1:L PR[91] R[100]mm/sec CNT100;
   1:  PR[91,1] = PR[90,1] + -33.883;
   1:  PR[91,2] = PR[90,2] + 0.428;
   1:  PR[91,3] = PR[90,3] + 26.258;
   1:L PR[91] R[100]mm/sec CNT100;
   1:  PR[91,1] = PR[90,1] + -33.859;
   1:  PR[91,2] = PR[90,2] + -0.516;
   1:  PR[91,3] = PR[90,3] + 26.265;
   1:L PR[91] R[100]mm/sec CNT100;
   1:  PR[91,1] = PR[90,1] + -33.795;
   1:  PR[91,2] = PR[90,2] + -1.359;
   1:  PR[91,3] = PR[90,3] + 26.272;
   1:L PR[91] R[100]mm/sec CNT100;
   1:  PR[91,1] = PR[90,1] + -33.678;
   1:  PR[91,2] = PR[90,2] + -2.249;
   1:  PR[91,3] = PR[90,3] + 26.278;
   1:L PR[91] R[100]mm/sec CNT100;
   1:  PR[91,1] = PR[90,1] + -33.550;
   1:  PR[91,2] = PR[90,2] + -2.942;
   1:  PR[91,3] = PR[90,3] + 26.285;
   1:L PR[91] R[100]mm/sec CNT100;
   1:  PR[91,1] = PR[90,1] + -33.314;
   1:  PR[91,2] = PR[90,2] + -3.918;
   1:  PR[91,3] = PR[90,3] + 26.290;
   1:L PR[91] R[100]mm/sec CNT100;
   1:  PR[91,1] = PR[90,1] + -33.086;
   1:  PR[91,2] = PR[90,2] + -4.678;
   1:  PR[91,3] = PR[90,3] + 26.297;
   1:L PR[91] R[100]mm/sec CNT100;
   1:  PR[91,1] = PR[90,1] + -32.825;
   1:  PR[91,2] = PR[90,2] + -5.416;
   1:  PR[91,3] = PR[90,3] + 26.303;
   1:L PR[91] R[100]mm/sec CNT100;
   1:  PR[91,1] = PR[90,1] + -32.440;
   1:  PR[91,2] = PR[90,2] + -6.346;
   1:  PR[91,3] = PR[90,3] + 26.309;
   1:L PR[91] R[100]mm/sec CNT100;
   1:  PR[91,1] = PR[90,1] + -32.102;
   1:  PR[91,2] = PR[90,2] + -7.066;
   1:  PR[91,3] = PR[90,3] + 26.316;
   1:L PR[91] R[100]mm/sec CNT100;
   1:  PR[91,1] = PR[90,1] + -31.747;
   1:  PR[91,2] = PR[90,2] + -7.745;
   1:  PR[91,3] = PR[90,3] + 26.322;
   1:L PR[91] R[100]mm/sec CNT100;
   1:  PR[91,1] = PR[90,1] + -31.185;
   1:  PR[91,2] = PR[90,2] + -8.695;
   1:  PR[91,3] = PR[90,3] + 26.328;
   1:L PR[91] R[100]mm/sec CNT100;
   1:  PR[91,1] = PR[90,1] + -30.782;
   1:  PR[91,2] = PR[90,2] + -9.307;
   1:  PR[91,3] = PR[90,3] + 26.336;
   1:L PR[91] R[100]mm/sec CNT100;
   1:  PR[91,1] = PR[90,1] + -30.379;
   1:  PR[91,2] = PR[90,2] + -9.866;
   1:  PR[91,3] = PR[90,3] + 26.341;
   1:L PR[91] R[100]mm/sec CNT100;
   1:  PR[91,1] = PR[90,1] + -29.640;
   1:  PR[91,2] = PR[90,2] + -10.784;
   1:  PR[91,3] = PR[90,3] + 26.347;
   1:L PR[91] R[100]mm/sec CNT100;
   1:  PR[91,1] = PR[90,1] + -29.218;
   1:  PR[91,2] = PR[90,2] + -11.256;
   1:  PR[91,3] = PR[90,3] + 26.355;
   1:L PR[91] R[100]mm/sec CNT100;
   1:  PR[91,1] = PR[90,1] + -28.788;
   1:  PR[91,2] = PR[90,2] + -11.704;
   1:  PR[91,3] = PR[90,3] + 26.360;
   1:L PR[91] R[100]mm/sec CNT100;
   1:  PR[91,1] = PR[90,1] + -28.363;
   1:  PR[91,2] = PR[90,2] + -12.117;
   1:  PR[91,3] = PR[90,3] + 26.365;
   1:L PR[91] R[100]mm/sec CNT100;
   1:  PR[91,1] = PR[90,1] + -27.884;
   1:  PR[91,2] = PR[90,2] + -12.553;
   1:  PR[91,3] = PR[90,3] + 26.369;
   1:L PR[91] R[100]mm/sec CNT100;
   1:  PR[91,1] = PR[90,1] + -26.948;
   1:  PR[91,2] = PR[90,2] + -13.322;
   1:  PR[91,3] = PR[90,3] + 26.374;
   1:L PR[91] R[100]mm/sec CNT100;
   1:  PR[91,1] = PR[90,1] + -26.383;
   1:  PR[91,2] = PR[90,2] + -13.741;
   1:  PR[91,3] = PR[90,3] + 26.383;
   1:L PR[91] R[100]mm/sec CNT100;
   1:  PR[91,1] = PR[90,1] + -25.769;
   1:  PR[91,2] = PR[90,2] + -14.160;
   1:  PR[91,3] = PR[90,3] + 26.388;
   1:L PR[91] R[100]mm/sec CNT100;
   1:  PR[91,1] = PR[90,1] + -24.753;
   1:  PR[91,2] = PR[90,2] + -14.785;
   1:  PR[91,3] = PR[90,3] + 26.393;
   1:L PR[91] R[100]mm/sec CNT100;
   1:  PR[91,1] = PR[90,1] + -23.755;
   1:  PR[91,2] = PR[90,2] + -15.318;
   1:  PR[91,3] = PR[90,3] + 26.402;
   1:L PR[91] R[100]mm/sec CNT100;
   1:  PR[91,1] = PR[90,1] + -22.778;
   1:  PR[91,2] = PR[90,2] + -15.770;
   1:  PR[91,3] = PR[90,3] + 26.411;
   1:L PR[91] R[100]mm/sec CNT100;
   1:  PR[91,1] = PR[90,1] + -22.013;
   1:  PR[91,2] = PR[90,2] + -16.085;
   1:  PR[91,3] = PR[90,3] + 26.419;
   1:L PR[91] R[100]mm/sec CNT100;
   1:  PR[91,1] = PR[90,1] + -21.189;
   1:  PR[91,2] = PR[90,2] + -16.381;
   1:  PR[91,3] = PR[90,3] + 26.425;
   1:L PR[91] R[100]mm/sec CNT100;
   1:  PR[91,1] = PR[90,1] + -20.300;
   1:  PR[91,2] = PR[90,2] + -16.655;
   1:  PR[91,3] = PR[90,3] + 26.431;
   1:L PR[91] R[100]mm/sec CNT100;
   1:  PR[91,1] = PR[90,1] + -19.288;
   1:  PR[91,2] = PR[90,2] + -16.913;
   1:  PR[91,3] = PR[90,3] + 26.438;
   1:L PR[91] R[100]mm/sec CNT100;
   1:  PR[91,1] = PR[90,1] + -18.316;
   1:  PR[91,2] = PR[90,2] + -17.110;
   1:  PR[91,3] = PR[90,3] + 26.446;
   1:L PR[91] R[100]mm/sec CNT100;
   1:  PR[91,1] = PR[90,1] + -17.332;
   1:  PR[91,2] = PR[90,2] + -17.261;
   1:  PR[91,3] = PR[90,3] + 26.453;
   1:L PR[91] R[100]mm/sec CNT100;
   1:  PR[91,1] = PR[90,1] + -16.341;
   1:  PR[91,2] = PR[90,2] + -17.364;
   1:  PR[91,3] = PR[90,3] + 26.460;
   1:L PR[91] R[100]mm/sec CNT100;
   1:  PR[91,1] = PR[90,1] + -15.344;
   1:  PR[91,2] = PR[90,2] + -17.418;
   1:  PR[91,3] = PR[90,3] + 26.468;
   1:L PR[91] R[100]mm/sec CNT100;
   1:  PR[91,1] = PR[90,1] + -14.345;
   1:  PR[91,2] = PR[90,2] + -17.423;
   1:  PR[91,3] = PR[90,3] + 26.475;
   1:L PR[91] R[100]mm/sec CNT100;
   1:  PR[91,1] = PR[90,1] + -13.345;
   1:  PR[91,2] = PR[90,2] + -17.379;
   1:  PR[91,3] = PR[90,3] + 26.483;
   1:L PR[91] R[100]mm/sec CNT100;
   1:  PR[91,1] = PR[90,1] + -12.822;
   1:  PR[91,2] = PR[90,2] + -17.331;
   1:  PR[91,3] = PR[90,3] + 26.490;
   1:L PR[91] R[100]mm/sec CNT100;
   1:  PR[91,1] = PR[90,1] + -12.351;
   1:  PR[91,2] = PR[90,2] + -17.285;
   1:  PR[91,3] = PR[90,3] + 26.494;
   1:L PR[91] R[100]mm/sec CNT100;
   1:  PR[91,1] = PR[90,1] + -11.359;
   1:  PR[91,2] = PR[90,2] + -17.141;
   1:  PR[91,3] = PR[90,3] + 26.497;
   1:L PR[91] R[100]mm/sec CNT100;
   1:  PR[91,1] = PR[90,1] + -10.378;
   1:  PR[91,2] = PR[90,2] + -16.948;
   1:  PR[91,3] = PR[90,3] + 26.505;
   1:L PR[91] R[100]mm/sec CNT100;
   1:  PR[91,1] = PR[90,1] + -9.410;
   1:  PR[91,2] = PR[90,2] + -16.706;
   1:  PR[91,3] = PR[90,3] + 26.512;
   1:L PR[91] R[100]mm/sec CNT100;
   1:  PR[91,1] = PR[90,1] + -8.290;
   1:  PR[91,2] = PR[90,2] + -16.357;
   1:  PR[91,3] = PR[90,3] + 26.520;
   1:L PR[91] R[100]mm/sec CNT100;
   1:  PR[91,1] = PR[90,1] + -7.514;
   1:  PR[91,2] = PR[90,2] + -16.076;
   1:  PR[91,3] = PR[90,3] + 26.528;
   1:L PR[91] R[100]mm/sec CNT100;
   1:  PR[91,1] = PR[90,1] + -6.594;
   1:  PR[91,2] = PR[90,2] + -15.689;
   1:  PR[91,3] = PR[90,3] + 26.534;
   1:L PR[91] R[100]mm/sec CNT100;
   1:  PR[91,1] = PR[90,1] + -5.691;
   1:  PR[91,2] = PR[90,2] + -15.255;
   1:  PR[91,3] = PR[90,3] + 26.542;
   1:L PR[91] R[100]mm/sec CNT100;
   1:  PR[91,1] = PR[90,1] + -4.804;
   1:  PR[91,2] = PR[90,2] + -14.772;
   1:  PR[91,3] = PR[90,3] + 26.549;
   1:L PR[91] R[100]mm/sec CNT100;
   1:  PR[91,1] = PR[90,1] + -3.950;
   1:  PR[91,2] = PR[90,2] + -14.247;
   1:  PR[91,3] = PR[90,3] + 26.557;
   1:L PR[91] R[100]mm/sec CNT100;
   1:  PR[91,1] = PR[90,1] + -3.128;
   1:  PR[91,2] = PR[90,2] + -13.680;
   1:  PR[91,3] = PR[90,3] + 26.564;
   1:L PR[91] R[100]mm/sec CNT100;
   1:  PR[91,1] = PR[90,1] + -2.487;
   1:  PR[91,2] = PR[90,2] + -13.189;
   1:  PR[91,3] = PR[90,3] + 26.571;
   1:L PR[91] R[100]mm/sec CNT100;
   1:  PR[91,1] = PR[90,1] + -2.021;
   1:  PR[91,2] = PR[90,2] + -12.801;
   1:  PR[91,3] = PR[90,3] + 26.577;
   1:L PR[91] R[100]mm/sec CNT100;
   1:  PR[91,1] = PR[90,1] + -1.644;
   1:  PR[91,2] = PR[90,2] + -12.523;
   1:  PR[91,3] = PR[90,3] + 26.582;
   1:L PR[91] R[100]mm/sec CNT100;
   1:  PR[91,1] = PR[90,1] + -1.206;
   1:  PR[91,2] = PR[90,2] + -12.304;
   1:  PR[91,3] = PR[90,3] + 26.585;
   1:L PR[91] R[100]mm/sec CNT100;
   1:  PR[91,1] = PR[90,1] + -0.967;
   1:  PR[91,2] = PR[90,2] + -12.225;
   1:  PR[91,3] = PR[90,3] + 26.589;
   1:L PR[91] R[100]mm/sec CNT100;
   1:  PR[91,1] = PR[90,1] + -0.723;
   1:  PR[91,2] = PR[90,2] + -12.155;
   1:  PR[91,3] = PR[90,3] + 26.591;
   1:L PR[91] R[100]mm/sec CNT100;
   1:  PR[91,1] = PR[90,1] + -0.239;
   1:  PR[91,2] = PR[90,2] + -12.094;
   1:  PR[91,3] = PR[90,3] + 26.593;
   1:L PR[91] R[100]mm/sec CNT100;
   1:  PR[91,1] = PR[90,1] + 0.256;
   1:  PR[91,2] = PR[90,2] + -12.116;
   1:  PR[91,3] = PR[90,3] + 26.596;
   1:L PR[91] R[100]mm/sec CNT100;
   1:  PR[91] = PR[90];
   1:  PR[91,1] = PR[90,1] + 0.840;
   1:  PR[91,2] = PR[90,2] + -12.856;
   1:  PR[91,3] = PR[90,3] + 27.930;
   1:L PR[91] R[100]mm/sec CNT100;
   1:  PR[91,1] = PR[90,1] + 1.300;
   1:  PR[91,2] = PR[90,2] + -13.063;
   1:  PR[91,3] = PR[90,3] + 26.604;
   1:L PR[91] R[100]mm/sec CNT100;
   1:  PR[91,1] = PR[90,1] + 1.701;
   1:  PR[91,2] = PR[90,2] + -13.334;
   1:  PR[91,3] = PR[90,3] + 26.608;
   1:L PR[91] R[100]mm/sec CNT100;
   1:  PR[91,1] = PR[90,1] + 2.162;
   1:  PR[91,2] = PR[90,2] + -13.692;
   1:  PR[91,3] = PR[90,3] + 26.611;
   1:L PR[91] R[100]mm/sec CNT100;
   1:  PR[91,1] = PR[90,1] + 2.968;
   1:  PR[91,2] = PR[90,2] + -14.260;
   1:  PR[91,3] = PR[90,3] + 26.615;
   1:L PR[91] R[100]mm/sec CNT100;
   1:  PR[91,1] = PR[90,1] + 3.805;
   1:  PR[91,2] = PR[90,2] + -14.788;
   1:  PR[91,3] = PR[90,3] + 26.623;
   1:L PR[91] R[100]mm/sec CNT100;
   1:  PR[91,1] = PR[90,1] + 4.259;
   1:  PR[91,2] = PR[90,2] + -15.046;
   1:  PR[91,3] = PR[90,3] + 26.630;
   1:L PR[91] R[100]mm/sec CNT100;
   1:  PR[91,1] = PR[90,1] + 4.664;
   1:  PR[91,2] = PR[90,2] + -15.268;
   1:  PR[91,3] = PR[90,3] + 26.634;
   1:L PR[91] R[100]mm/sec CNT100;
   1:  PR[91,1] = PR[90,1] + 5.555;
   1:  PR[91,2] = PR[90,2] + -15.708;
   1:  PR[91,3] = PR[90,3] + 26.638;
   1:L PR[91] R[100]mm/sec CNT100;
   1:  PR[91,1] = PR[90,1] + 6.467;
   1:  PR[91,2] = PR[90,2] + -16.102;
   1:  PR[91,3] = PR[90,3] + 26.645;
   1:L PR[91] R[100]mm/sec CNT100;
   1:  PR[91,1] = PR[90,1] + 7.396;
   1:  PR[91,2] = PR[90,2] + -16.450;
   1:  PR[91,3] = PR[90,3] + 26.653;
   1:L PR[91] R[100]mm/sec CNT100;
   1:  PR[91,1] = PR[90,1] + 8.555;
   1:  PR[91,2] = PR[90,2] + -16.809;
   1:  PR[91,3] = PR[90,3] + 26.660;
   1:L PR[91] R[100]mm/sec CNT100;
   1:  PR[91,1] = PR[90,1] + 9.309;
   1:  PR[91,2] = PR[90,2] + -17.006;
   1:  PR[91,3] = PR[90,3] + 26.669;
   1:L PR[91] R[100]mm/sec CNT100;
   1:  PR[91,1] = PR[90,1] + 10.285;
   1:  PR[91,2] = PR[90,2] + -17.211;
   1:  PR[91,3] = PR[90,3] + 26.675;
   1:L PR[91] R[100]mm/sec CNT100;
   1:  PR[91,1] = PR[90,1] + 11.270;
   1:  PR[91,2] = PR[90,2] + -17.368;
   1:  PR[91,3] = PR[90,3] + 26.682;
   1:L PR[91] R[100]mm/sec CNT100;
   1:  PR[91,1] = PR[90,1] + 12.271;
   1:  PR[91,2] = PR[90,2] + -17.478;
   1:  PR[91,3] = PR[90,3] + 26.690;
   1:L PR[91] R[100]mm/sec CNT100;
   1:  PR[91,1] = PR[90,1] + 13.281;
   1:  PR[91,2] = PR[90,2] + -17.538;
   1:  PR[91,3] = PR[90,3] + 26.697;
   1:L PR[91] R[100]mm/sec CNT100;
   1:  PR[91,1] = PR[90,1] + 14.069;
   1:  PR[91,2] = PR[90,2] + -17.549;
   1:  PR[91,3] = PR[90,3] + 26.705;
   1:L PR[91] R[100]mm/sec CNT100;
   1:  PR[91,1] = PR[90,1] + 15.009;
   1:  PR[91,2] = PR[90,2] + -17.523;
   1:  PR[91,3] = PR[90,3] + 26.711;
   1:L PR[91] R[100]mm/sec CNT100;
   1:  PR[91,1] = PR[90,1] + 15.947;
   1:  PR[91,2] = PR[90,2] + -17.454;
   1:  PR[91,3] = PR[90,3] + 26.718;
   1:L PR[91] R[100]mm/sec CNT100;
   1:  PR[91,1] = PR[90,1] + 16.881;
   1:  PR[91,2] = PR[90,2] + -17.341;
   1:  PR[91,3] = PR[90,3] + 26.725;
   1:L PR[91] R[100]mm/sec CNT100;
   1:  PR[91,1] = PR[90,1] + 17.811;
   1:  PR[91,2] = PR[90,2] + -17.185;
   1:  PR[91,3] = PR[90,3] + 26.732;
   1:L PR[91] R[100]mm/sec CNT100;
   1:  PR[91,1] = PR[90,1] + 18.734;
   1:  PR[91,2] = PR[90,2] + -16.985;
   1:  PR[91,3] = PR[90,3] + 26.739;
   1:L PR[91] R[100]mm/sec CNT100;
   1:  PR[91,1] = PR[90,1] + 19.647;
   1:  PR[91,2] = PR[90,2] + -16.742;
   1:  PR[91,3] = PR[90,3] + 26.746;
   1:L PR[91] R[100]mm/sec CNT100;
   1:  PR[91,1] = PR[90,1] + 20.548;
   1:  PR[91,2] = PR[90,2] + -16.456;
   1:  PR[91,3] = PR[90,3] + 26.753;
   1:L PR[91] R[100]mm/sec CNT100;
   1:  PR[91,1] = PR[90,1] + 21.436;
   1:  PR[91,2] = PR[90,2] + -16.128;
   1:  PR[91,3] = PR[90,3] + 26.760;
   1:L PR[91] R[100]mm/sec CNT100;
   1:  PR[91,1] = PR[90,1] + 22.307;
   1:  PR[91,2] = PR[90,2] + -15.759;
   1:  PR[91,3] = PR[90,3] + 26.767;
   1:L PR[91] R[100]mm/sec CNT100;
   1:  PR[91,1] = PR[90,1] + 23.160;
   1:  PR[91,2] = PR[90,2] + -15.349;
   1:  PR[91,3] = PR[90,3] + 26.774;
   1:L PR[91] R[100]mm/sec CNT100;
   1:  PR[91,1] = PR[90,1] + 24.016;
   1:  PR[91,2] = PR[90,2] + -14.889;
   1:  PR[91,3] = PR[90,3] + 26.781;
   1:L PR[91] R[100]mm/sec CNT100;
   1:  PR[91,1] = PR[90,1] + 24.808;
   1:  PR[91,2] = PR[90,2] + -14.412;
   1:  PR[91,3] = PR[90,3] + 26.789;
   1:L PR[91] R[100]mm/sec CNT100;
   1:  PR[91,1] = PR[90,1] + 25.647;
   1:  PR[91,2] = PR[90,2] + -13.847;
   1:  PR[91,3] = PR[90,3] + 26.796;
   1:L PR[91] R[100]mm/sec CNT100;
   1:  PR[91,1] = PR[90,1] + 26.341;
   1:  PR[91,2] = PR[90,2] + -13.329;
   1:  PR[91,3] = PR[90,3] + 26.803;
   1:L PR[91] R[100]mm/sec CNT100;
   1:  PR[91,1] = PR[90,1] + 27.146;
   1:  PR[91,2] = PR[90,2] + -12.663;
   1:  PR[91,3] = PR[90,3] + 26.810;
   1:L PR[91] R[100]mm/sec CNT100;
   1:  PR[91,1] = PR[90,1] + 27.745;
   1:  PR[91,2] = PR[90,2] + -12.112;
   1:  PR[91,3] = PR[90,3] + 26.818;
   1:L PR[91] R[100]mm/sec CNT100;
   1:  PR[91,1] = PR[90,1] + 28.498;
   1:  PR[91,2] = PR[90,2] + -11.346;
   1:  PR[91,3] = PR[90,3] + 26.824;
   1:L PR[91] R[100]mm/sec CNT100;
   1:  PR[91,1] = PR[90,1] + 29.004;
   1:  PR[91,2] = PR[90,2] + -10.773;
   1:  PR[91,3] = PR[90,3] + 26.832;
   1:L PR[91] R[100]mm/sec CNT100;
   1:  PR[91,1] = PR[90,1] + 29.700;
   1:  PR[91,2] = PR[90,2] + -9.901;
   1:  PR[91,3] = PR[90,3] + 26.837;
   1:L PR[91] R[100]mm/sec CNT100;
   1:  PR[91,1] = PR[90,1] + 30.127;
   1:  PR[91,2] = PR[90,2] + -9.304;
   1:  PR[91,3] = PR[90,3] + 26.846;
   1:L PR[91] R[100]mm/sec CNT100;
   1:  PR[91,1] = PR[90,1] + 30.756;
   1:  PR[91,2] = PR[90,2] + -8.324;
   1:  PR[91,3] = PR[90,3] + 26.851;
   1:L PR[91] R[100]mm/sec CNT100;
   1:  PR[91,1] = PR[90,1] + 31.105;
   1:  PR[91,2] = PR[90,2] + -7.713;
   1:  PR[91,3] = PR[90,3] + 26.860;
   1:L PR[91] R[100]mm/sec CNT100;
   1:  PR[91,1] = PR[90,1] + 31.649;
   1:  PR[91,2] = PR[90,2] + -6.642;
   1:  PR[91,3] = PR[90,3] + 26.865;
   1:L PR[91] R[100]mm/sec CNT100;
   1:  PR[91,1] = PR[90,1] + 31.924;
   1:  PR[91,2] = PR[90,2] + -6.022;
   1:  PR[91,3] = PR[90,3] + 26.874;
   1:L PR[91] R[100]mm/sec CNT100;
   1:  PR[91,1] = PR[90,1] + 32.122;
   1:  PR[91,2] = PR[90,2] + -5.534;
   1:  PR[91,3] = PR[90,3] + 26.879;
   1:L PR[91] R[100]mm/sec CNT100;
   1:  PR[91,1] = PR[90,1] + 32.347;
   1:  PR[91,2] = PR[90,2] + -4.920;
   1:  PR[91,3] = PR[90,3] + 26.883;
   1:L PR[91] R[100]mm/sec CNT100;
   1:  PR[91,1] = PR[90,1] + 32.539;
   1:  PR[91,2] = PR[90,2] + -4.324;
   1:  PR[91,3] = PR[90,3] + 26.888;
   1:L PR[91] R[100]mm/sec CNT100;
   1:  PR[91,1] = PR[90,1] + 32.684;
   1:  PR[91,2] = PR[90,2] + -3.813;
   1:  PR[91,3] = PR[90,3] + 26.893;
   1:L PR[91] R[100]mm/sec CNT100;
   1:  PR[91,1] = PR[90,1] + 32.829;
   1:  PR[91,2] = PR[90,2] + -3.220;
   1:  PR[91,3] = PR[90,3] + 26.897;
   1:L PR[91] R[100]mm/sec CNT100;
   1:  PR[91,1] = PR[90,1] + 32.949;
   1:  PR[91,2] = PR[90,2] + -2.627;
   1:  PR[91,3] = PR[90,3] + 26.901;
   1:L PR[91] R[100]mm/sec CNT100;
   1:  PR[91,1] = PR[90,1] + 33.041;
   1:  PR[91,2] = PR[90,2] + -2.071;
   1:  PR[91,3] = PR[90,3] + 26.906;
   1:L PR[91] R[100]mm/sec CNT100;
   1:  PR[91,1] = PR[90,1] + 33.118;
   1:  PR[91,2] = PR[90,2] + -1.457;
   1:  PR[91,3] = PR[90,3] + 26.910;
   1:L PR[91] R[100]mm/sec CNT100;
   1:  PR[91,1] = PR[90,1] + 33.173;
   1:  PR[91,2] = PR[90,2] + -0.833;
   1:  PR[91,3] = PR[90,3] + 26.915;
   1:L PR[91] R[100]mm/sec CNT100;
   1:  PR[91,1] = PR[90,1] + 33.204;
   1:  PR[91,2] = PR[90,2] + -0.227;
   1:  PR[91,3] = PR[90,3] + 26.919;
   1:L PR[91] R[100]mm/sec CNT100;
   1:  PR[91,1] = PR[90,1] + 33.215;
   1:  PR[91,2] = PR[90,2] + 0.428;
   1:  PR[91,3] = PR[90,3] + 26.924;
   1:L PR[91] R[100]mm/sec CNT100;
   1:  PR[91,1] = PR[90,1] + 33.204;
   1:  PR[91,2] = PR[90,2] + 1.082;
   1:  PR[91,3] = PR[90,3] + 26.929;
   1:L PR[91] R[100]mm/sec CNT100;
   1:  PR[91,1] = PR[90,1] + 33.173;
   1:  PR[91,2] = PR[90,2] + 1.688;
   1:  PR[91,3] = PR[90,3] + 26.934;
   1:L PR[91] R[100]mm/sec CNT100;
   1:  PR[91,1] = PR[90,1] + 33.118;
   1:  PR[91,2] = PR[90,2] + 2.312;
   1:  PR[91,3] = PR[90,3] + 26.938;
   1:L PR[91] R[100]mm/sec CNT100;
   1:  PR[91,1] = PR[90,1] + 33.041;
   1:  PR[91,2] = PR[90,2] + 2.927;
   1:  PR[91,3] = PR[90,3] + 26.943;
   1:L PR[91] R[100]mm/sec CNT100;
   1:  PR[91,1] = PR[90,1] + 32.949;
   1:  PR[91,2] = PR[90,2] + 3.482;
   1:  PR[91,3] = PR[90,3] + 26.948;
   1:L PR[91] R[100]mm/sec CNT100;
   1:  PR[91,1] = PR[90,1] + 32.829;
   1:  PR[91,2] = PR[90,2] + 4.075;
   1:  PR[91,3] = PR[90,3] + 26.952;
   1:L PR[91] R[100]mm/sec CNT100;
   1:  PR[91,1] = PR[90,1] + 32.684;
   1:  PR[91,2] = PR[90,2] + 4.668;
   1:  PR[91,3] = PR[90,3] + 26.956;
   1:L PR[91] R[100]mm/sec CNT100;
   1:  PR[91,1] = PR[90,1] + 32.539;
   1:  PR[91,2] = PR[90,2] + 5.179;
   1:  PR[91,3] = PR[90,3] + 26.961;
   1:L PR[91] R[100]mm/sec CNT100;
   1:  PR[91,1] = PR[90,1] + 32.347;
   1:  PR[91,2] = PR[90,2] + 5.775;
   1:  PR[91,3] = PR[90,3] + 26.965;
   1:L PR[91] R[100]mm/sec CNT100;
   1:  PR[91,1] = PR[90,1] + 32.122;
   1:  PR[91,2] = PR[90,2] + 6.389;
   1:  PR[91,3] = PR[90,3] + 26.970;
   1:L PR[91] R[100]mm/sec CNT100;
   1:  PR[91,1] = PR[90,1] + 31.924;
   1:  PR[91,2] = PR[90,2] + 6.877;
   1:  PR[91,3] = PR[90,3] + 26.975;
   1:L PR[91] R[100]mm/sec CNT100;
   1:  PR[91,1] = PR[90,1] + 31.649;
   1:  PR[91,2] = PR[90,2] + 7.497;
   1:  PR[91,3] = PR[90,3] + 26.979;
   1:L PR[91] R[100]mm/sec CNT100;
   1:  PR[91,1] = PR[90,1] + 31.105;
   1:  PR[91,2] = PR[90,2] + 8.568;
   1:  PR[91,3] = PR[90,3] + 26.984;
   1:L PR[91] R[100]mm/sec CNT100;
   1:  PR[91,1] = PR[90,1] + 30.756;
   1:  PR[91,2] = PR[90,2] + 9.179;
   1:  PR[91,3] = PR[90,3] + 26.993;
   1:L PR[91] R[100]mm/sec CNT100;
   1:  PR[91,1] = PR[90,1] + 30.127;
   1:  PR[91,2] = PR[90,2] + 10.159;
   1:  PR[91,3] = PR[90,3] + 26.998;
   1:L PR[91] R[100]mm/sec CNT100;
   1:  PR[91,1] = PR[90,1] + 29.700;
   1:  PR[91,2] = PR[90,2] + 10.756;
   1:  PR[91,3] = PR[90,3] + 27.007;
   1:L PR[91] R[100]mm/sec CNT100;
   1:  PR[91,1] = PR[90,1] + 29.004;
   1:  PR[91,2] = PR[90,2] + 11.628;
   1:  PR[91,3] = PR[90,3] + 27.012;
   1:L PR[91] R[100]mm/sec CNT100;
   1:  PR[91,1] = PR[90,1] + 28.498;
   1:  PR[91,2] = PR[90,2] + 12.201;
   1:  PR[91,3] = PR[90,3] + 27.020;
   1:L PR[91] R[100]mm/sec CNT100;
   1:  PR[91,1] = PR[90,1] + 27.744;
   1:  PR[91,2] = PR[90,2] + 12.968;
   1:  PR[91,3] = PR[90,3] + 27.026;
   1:L PR[91] R[100]mm/sec CNT100;
   1:  PR[91,1] = PR[90,1] + 27.146;
   1:  PR[91,2] = PR[90,2] + 13.518;
   1:  PR[91,3] = PR[90,3] + 27.034;
   1:L PR[91] R[100]mm/sec CNT100;
   1:  PR[91,1] = PR[90,1] + 26.341;
   1:  PR[91,2] = PR[90,2] + 14.184;
   1:  PR[91,3] = PR[90,3] + 27.040;
   1:L PR[91] R[100]mm/sec CNT100;
   1:  PR[91,1] = PR[90,1] + 25.647;
   1:  PR[91,2] = PR[90,2] + 14.703;
   1:  PR[91,3] = PR[90,3] + 27.048;
   1:L PR[91] R[100]mm/sec CNT100;
   1:  PR[91,1] = PR[90,1] + 24.807;
   1:  PR[91,2] = PR[90,2] + 15.267;
   1:  PR[91,3] = PR[90,3] + 27.055;
   1:L PR[91] R[100]mm/sec CNT100;
   1:  PR[91,1] = PR[90,1] + 24.016;
   1:  PR[91,2] = PR[90,2] + 15.744;
   1:  PR[91,3] = PR[90,3] + 27.062;
   1:L PR[91] R[100]mm/sec CNT100;
   1:  PR[91,1] = PR[90,1] + 23.151;
   1:  PR[91,2] = PR[90,2] + 16.209;
   1:  PR[91,3] = PR[90,3] + 27.069;
   1:L PR[91] R[100]mm/sec CNT100;
   1:  PR[91,1] = PR[90,1] + 22.307;
   1:  PR[91,2] = PR[90,2] + 16.614;
   1:  PR[91,3] = PR[90,3] + 27.076;
   1:L PR[91] R[100]mm/sec CNT100;
   1:  PR[91,1] = PR[90,1] + 21.435;
   1:  PR[91,2] = PR[90,2] + 16.983;
   1:  PR[91,3] = PR[90,3] + 27.083;
   1:L PR[91] R[100]mm/sec CNT100;
   1:  PR[91,1] = PR[90,1] + 20.548;
   1:  PR[91,2] = PR[90,2] + 17.311;
   1:  PR[91,3] = PR[90,3] + 27.091;
   1:L PR[91] R[100]mm/sec CNT100;
   1:  PR[91,1] = PR[90,1] + 19.646;
   1:  PR[91,2] = PR[90,2] + 17.597;
   1:  PR[91,3] = PR[90,3] + 27.098;
   1:L PR[91] R[100]mm/sec CNT100;
   1:  PR[91,1] = PR[90,1] + 18.733;
   1:  PR[91,2] = PR[90,2] + 17.840;
   1:  PR[91,3] = PR[90,3] + 27.105;
   1:L PR[91] R[100]mm/sec CNT100;
   1:  PR[91,1] = PR[90,1] + 17.811;
   1:  PR[91,2] = PR[90,2] + 18.040;
   1:  PR[91,3] = PR[90,3] + 27.112;
   1:L PR[91] R[100]mm/sec CNT100;
   1:  PR[91,1] = PR[90,1] + 16.881;
   1:  PR[91,2] = PR[90,2] + 18.196;
   1:  PR[91,3] = PR[90,3] + 27.119;
   1:L PR[91] R[100]mm/sec CNT100;
   1:  PR[91,1] = PR[90,1] + 15.944;
   1:  PR[91,2] = PR[90,2] + 18.310;
   1:  PR[91,3] = PR[90,3] + 27.126;
   1:L PR[91] R[100]mm/sec CNT100;
   1:  PR[91,1] = PR[90,1] + 15.313;
   1:  PR[91,2] = PR[90,2] + 18.361;
   1:  PR[91,3] = PR[90,3] + 27.133;
   1:L PR[91] R[100]mm/sec CNT100;
   1:  PR[91,1] = PR[90,1] + 14.295;
   1:  PR[91,2] = PR[90,2] + 18.403;
   1:  PR[91,3] = PR[90,3] + 27.138;
   1:L PR[91] R[100]mm/sec CNT100;
   1:  PR[91,1] = PR[90,1] + 13.130;
   1:  PR[91,2] = PR[90,2] + 18.387;
   1:  PR[91,3] = PR[90,3] + 27.145;
   1:L PR[91] R[100]mm/sec CNT100;
   1:  PR[91,1] = PR[90,1] + 12.272;
   1:  PR[91,2] = PR[90,2] + 18.333;
   1:  PR[91,3] = PR[90,3] + 27.154;
   1:L PR[91] R[100]mm/sec CNT100;
   1:  PR[91,1] = PR[90,1] + 11.269;
   1:  PR[91,2] = PR[90,2] + 18.223;
   1:  PR[91,3] = PR[90,3] + 27.160;
   1:L PR[91] R[100]mm/sec CNT100;
   1:  PR[91,1] = PR[90,1] + 10.285;
   1:  PR[91,2] = PR[90,2] + 18.066;
   1:  PR[91,3] = PR[90,3] + 27.168;
   1:L PR[91] R[100]mm/sec CNT100;
   1:  PR[91,1] = PR[90,1] + 9.311;
   1:  PR[91,2] = PR[90,2] + 17.861;
   1:  PR[91,3] = PR[90,3] + 27.175;
   1:L PR[91] R[100]mm/sec CNT100;
   1:  PR[91,1] = PR[90,1] + 8.347;
   1:  PR[91,2] = PR[90,2] + 17.607;
   1:  PR[91,3] = PR[90,3] + 27.183;
   1:L PR[91] R[100]mm/sec CNT100;
   1:  PR[91,1] = PR[90,1] + 7.399;
   1:  PR[91,2] = PR[90,2] + 17.306;
   1:  PR[91,3] = PR[90,3] + 27.190;
   1:L PR[91] R[100]mm/sec CNT100;
   1:  PR[91,1] = PR[90,1] + 6.466;
   1:  PR[91,2] = PR[90,2] + 16.957;
   1:  PR[91,3] = PR[90,3] + 27.198;
   1:L PR[91] R[100]mm/sec CNT100;
   1:  PR[91,1] = PR[90,1] + 5.555;
   1:  PR[91,2] = PR[90,2] + 16.563;
   1:  PR[91,3] = PR[90,3] + 27.205;
   1:L PR[91] R[100]mm/sec CNT100;
   1:  PR[91,1] = PR[90,1] + 4.663;
   1:  PR[91,2] = PR[90,2] + 16.123;
   1:  PR[91,3] = PR[90,3] + 27.213;
   1:L PR[91] R[100]mm/sec CNT100;
   1:  PR[91,1] = PR[90,1] + 4.259;
   1:  PR[91,2] = PR[90,2] + 15.902;
   1:  PR[91,3] = PR[90,3] + 27.220;
   1:L PR[91] R[100]mm/sec CNT100;
   1:  PR[91,1] = PR[90,1] + 3.805;
   1:  PR[91,2] = PR[90,2] + 15.642;
   1:  PR[91,3] = PR[90,3] + 27.224;
   1:L PR[91] R[100]mm/sec CNT100;
   1:  PR[91,1] = PR[90,1] + 2.967;
   1:  PR[91,2] = PR[90,2] + 15.115;
   1:  PR[91,3] = PR[90,3] + 27.228;
   1:L PR[91] R[100]mm/sec CNT100;
   1:  PR[91,1] = PR[90,1] + 2.163;
   1:  PR[91,2] = PR[90,2] + 14.548;
   1:  PR[91,3] = PR[90,3] + 27.235;
   1:L PR[91] R[100]mm/sec CNT100;
   1:  PR[91,1] = PR[90,1] + 1.698;
   1:  PR[91,2] = PR[90,2] + 14.187;
   1:  PR[91,3] = PR[90,3] + 27.242;
   1:L PR[91] R[100]mm/sec CNT100;
   1:  PR[91,1] = PR[90,1] + 1.300;
   1:  PR[91,2] = PR[90,2] + 13.918;
   1:  PR[91,3] = PR[90,3] + 27.247;
   1:L PR[91] R[100]mm/sec CNT100;
   1:  PR[91,1] = PR[90,1] + 0.840;
   1:  PR[91,2] = PR[90,2] + 13.711;
   1:  PR[91,3] = PR[90,3] + 27.250;
   1:L PR[91] R[100]mm/sec CNT100;
   1:  PR[91,1] = PR[90,1] + 0.357;
   1:  PR[91,2] = PR[90,2] + 13.588;
   1:  PR[91,3] = PR[90,3] + 27.254;
   1:L PR[91] R[100]mm/sec CNT100;
   1:  PR[91,1] = PR[90,1] + -0.137;
   1:  PR[91,2] = PR[90,2] + 13.547;
   1:  PR[91,3] = PR[90,3] + 27.258;
   1:L PR[91] R[100]mm/sec CNT100;
   1:  PR[91,1] = PR[90,1] + -0.621;
   1:  PR[91,2] = PR[90,2] + 13.592;
   1:  PR[91,3] = PR[90,3] + 27.262;
   1:L PR[91] R[100]mm/sec CNT100;
   1:  PR[91,1] = PR[90,1] + -0.782;
   1:  PR[91,2] = PR[90,2] + 13.631;
   1:  PR[91,3] = PR[90,3] + 27.265;
   1:L PR[91] R[100]mm/sec CNT100;
   1:  PR[91,1] = PR[90,1] + -1.107;
   1:  PR[91,2] = PR[90,2] + 13.721;
   1:  PR[91,3] = PR[90,3] + 27.266;
   1:L PR[91] R[100]mm/sec CNT100;
   1:  PR[91,1] = PR[90,1] + -1.555;
   1:  PR[91,2] = PR[90,2] + 13.925;
   1:  PR[91,3] = PR[90,3] + 27.269;
   1:L PR[91] R[100]mm/sec CNT100;
   1:  PR[91,1] = PR[90,1] + -1.942;
   1:  PR[91,2] = PR[90,2] + 14.188;
   1:  PR[91,3] = PR[90,3] + 27.273;
   1:L PR[91] R[100]mm/sec CNT100;
   1:  PR[91,1] = PR[90,1] + -2.416;
   1:  PR[91,2] = PR[90,2] + 14.555;
   1:  PR[91,3] = PR[90,3] + 27.276;
   1:L PR[91] R[100]mm/sec CNT100;
   1:  PR[91,1] = PR[90,1] + -2.931;
   1:  PR[91,2] = PR[90,2] + 14.923;
   1:  PR[91,3] = PR[90,3] + 27.281;
   1:L PR[91] R[100]mm/sec CNT100;
   1:  PR[91,1] = PR[90,1] + -3.224;
   1:  PR[91,2] = PR[90,2] + 15.124;
   1:  PR[91,3] = PR[90,3] + 27.285;
   1:L PR[91] R[100]mm/sec CNT100;
   1:  PR[91,1] = PR[90,1] + -4.075;
   1:  PR[91,2] = PR[90,2] + 15.658;
   1:  PR[91,3] = PR[90,3] + 27.288;
   1:L PR[91] R[100]mm/sec CNT100;
   1:  PR[91,1] = PR[90,1] + -4.954;
   1:  PR[91,2] = PR[90,2] + 16.148;
   1:  PR[91,3] = PR[90,3] + 27.296;
   1:L PR[91] R[100]mm/sec CNT100;
   1:  PR[91,1] = PR[90,1] + -5.867;
   1:  PR[91,2] = PR[90,2] + 16.596;
   1:  PR[91,3] = PR[90,3] + 27.303;
   1:L PR[91] R[100]mm/sec CNT100;
   1:  PR[91,1] = PR[90,1] + -6.231;
   1:  PR[91,2] = PR[90,2] + 16.758;
   1:  PR[91,3] = PR[90,3] + 27.311;
   1:L PR[91] R[100]mm/sec CNT100;
   1:  PR[91,1] = PR[90,1] + -6.795;
   1:  PR[91,2] = PR[90,2] + 16.994;
   1:  PR[91,3] = PR[90,3] + 27.314;
   1:L PR[91] R[100]mm/sec CNT100;
   1:  PR[91,1] = PR[90,1] + -7.755;
   1:  PR[91,2] = PR[90,2] + 17.347;
   1:  PR[91,3] = PR[90,3] + 27.318;
   1:L PR[91] R[100]mm/sec CNT100;
   1:  PR[91,1] = PR[90,1] + -8.735;
   1:  PR[91,2] = PR[90,2] + 17.651;
   1:  PR[91,3] = PR[90,3] + 27.326;
   1:L PR[91] R[100]mm/sec CNT100;
   1:  PR[91,1] = PR[90,1] + -9.732;
   1:  PR[91,2] = PR[90,2] + 17.904;
   1:  PR[91,3] = PR[90,3] + 27.334;
   1:L PR[91] R[100]mm/sec CNT100;
   1:  PR[91,1] = PR[90,1] + -10.805;
   1:  PR[91,2] = PR[90,2] + 18.116;
   1:  PR[91,3] = PR[90,3] + 27.341;
   1:L PR[91] R[100]mm/sec CNT100;
   1:  PR[91,1] = PR[90,1] + -11.766;
   1:  PR[91,2] = PR[90,2] + 18.256;
   1:  PR[91,3] = PR[90,3] + 27.349;
   1:L PR[91] R[100]mm/sec CNT100;
   1:  PR[91,1] = PR[90,1] + -12.769;
   1:  PR[91,2] = PR[90,2] + 18.353;
   1:  PR[91,3] = PR[90,3] + 27.357;
   1:L PR[91] R[100]mm/sec CNT100;
   1:  PR[91,1] = PR[90,1] + -13.774;
   1:  PR[91,2] = PR[90,2] + 18.401;
   1:  PR[91,3] = PR[90,3] + 27.364;
   1:L PR[91] R[100]mm/sec CNT100;
   1:  PR[91,1] = PR[90,1] + -14.780;
   1:  PR[91,2] = PR[90,2] + 18.398;
   1:  PR[91,3] = PR[90,3] + 27.372;
   1:L PR[91] R[100]mm/sec CNT100;
   1:  PR[91,1] = PR[90,1] + -15.783;
   1:  PR[91,2] = PR[90,2] + 18.346;
   1:  PR[91,3] = PR[90,3] + 27.379;
   1:L PR[91] R[100]mm/sec CNT100;
   1:  PR[91,1] = PR[90,1] + -16.399;
   1:  PR[91,2] = PR[90,2] + 18.284;
   1:  PR[91,3] = PR[90,3] + 27.387;
   1:L PR[91] R[100]mm/sec CNT100;
   1:  PR[91,1] = PR[90,1] + -16.780;
   1:  PR[91,2] = PR[90,2] + 18.244;
   1:  PR[91,3] = PR[90,3] + 27.392;
   1:L PR[91] R[100]mm/sec CNT100;
   1:  PR[91,1] = PR[90,1] + -17.770;
   1:  PR[91,2] = PR[90,2] + 18.093;
   1:  PR[91,3] = PR[90,3] + 27.394;
   1:L PR[91] R[100]mm/sec CNT100;
   1:  PR[91,1] = PR[90,1] + -18.749;
   1:  PR[91,2] = PR[90,2] + 17.895;
   1:  PR[91,3] = PR[90,3] + 27.402;
   1:L PR[91] R[100]mm/sec CNT100;
   1:  PR[91,1] = PR[90,1] + -19.714;
   1:  PR[91,2] = PR[90,2] + 17.649;
   1:  PR[91,3] = PR[90,3] + 27.409;
   1:L PR[91] R[100]mm/sec CNT100;
   1:  PR[91,1] = PR[90,1] + -20.663;
   1:  PR[91,2] = PR[90,2] + 17.356;
   1:  PR[91,3] = PR[90,3] + 27.417;
   1:L PR[91] R[100]mm/sec CNT100;
   1:  PR[91,1] = PR[90,1] + -21.593;
   1:  PR[91,2] = PR[90,2] + 17.018;
   1:  PR[91,3] = PR[90,3] + 27.424;
   1:L PR[91] R[100]mm/sec CNT100;
   1:  PR[91,1] = PR[90,1] + -22.502;
   1:  PR[91,2] = PR[90,2] + 16.635;
   1:  PR[91,3] = PR[90,3] + 27.432;
   1:L PR[91] R[100]mm/sec CNT100;
   1:  PR[91,1] = PR[90,1] + -23.397;
   1:  PR[91,2] = PR[90,2] + 16.204;
   1:  PR[91,3] = PR[90,3] + 27.439;
   1:L PR[91] R[100]mm/sec CNT100;
   1:  PR[91,1] = PR[90,1] + -24.250;
   1:  PR[91,2] = PR[90,2] + 15.744;
   1:  PR[91,3] = PR[90,3] + 27.446;
   1:L PR[91] R[100]mm/sec CNT100;
   1:  PR[91,1] = PR[90,1] + -25.126;
   1:  PR[91,2] = PR[90,2] + 15.213;
   1:  PR[91,3] = PR[90,3] + 27.454;
   1:L PR[91] R[100]mm/sec CNT100;
   1:  PR[91,1] = PR[90,1] + -25.889;
   1:  PR[91,2] = PR[90,2] + 14.697;
   1:  PR[91,3] = PR[90,3] + 27.461;
   1:L PR[91] R[100]mm/sec CNT100;
   1:  PR[91,1] = PR[90,1] + -26.587;
   1:  PR[91,2] = PR[90,2] + 14.175;
   1:  PR[91,3] = PR[90,3] + 27.468;
   1:L PR[91] R[100]mm/sec CNT100;
   1:  PR[91,1] = PR[90,1] + -27.397;
   1:  PR[91,2] = PR[90,2] + 13.505;
   1:  PR[91,3] = PR[90,3] + 27.475;
   1:L PR[91] R[100]mm/sec CNT100;
   1:  PR[91,1] = PR[90,1] + -28.196;
   1:  PR[91,2] = PR[90,2] + 12.761;
   1:  PR[91,3] = PR[90,3] + 27.483;
   1:L PR[91] R[100]mm/sec CNT100;
   1:  PR[91,1] = PR[90,1] + -28.755;
   1:  PR[91,2] = PR[90,2] + 12.184;
   1:  PR[91,3] = PR[90,3] + 27.491;
   1:L PR[91] R[100]mm/sec CNT100;
   1:  PR[91,1] = PR[90,1] + -29.264;
   1:  PR[91,2] = PR[90,2] + 11.610;
   1:  PR[91,3] = PR[90,3] + 27.497;
   1:L PR[91] R[100]mm/sec CNT100;
   1:  PR[91,1] = PR[90,1] + -29.956;
   1:  PR[91,2] = PR[90,2] + 10.743;
   1:  PR[91,3] = PR[90,3] + 27.503;
   1:L PR[91] R[100]mm/sec CNT100;
   1:  PR[91,1] = PR[90,1] + -30.618;
   1:  PR[91,2] = PR[90,2] + 9.792;
   1:  PR[91,3] = PR[90,3] + 27.511;
   1:L PR[91] R[100]mm/sec CNT100;
   1:  PR[91,1] = PR[90,1] + -31.003;
   1:  PR[91,2] = PR[90,2] + 9.174;
   1:  PR[91,3] = PR[90,3] + 27.520;
   1:L PR[91] R[100]mm/sec CNT100;
   1:  PR[91,1] = PR[90,1] + -31.351;
   1:  PR[91,2] = PR[90,2] + 8.560;
   1:  PR[91,3] = PR[90,3] + 27.525;
   1:L PR[91] R[100]mm/sec CNT100;
   1:  PR[91,1] = PR[90,1] + -31.896;
   1:  PR[91,2] = PR[90,2] + 7.476;
   1:  PR[91,3] = PR[90,3] + 27.530;
   1:L PR[91] R[100]mm/sec CNT100;
   1:  PR[91,1] = PR[90,1] + -32.172;
   1:  PR[91,2] = PR[90,2] + 6.845;
   1:  PR[91,3] = PR[90,3] + 27.539;
   1:L PR[91] R[100]mm/sec CNT100;
   1:  PR[91,1] = PR[90,1] + -32.418;
   1:  PR[91,2] = PR[90,2] + 6.224;
   1:  PR[91,3] = PR[90,3] + 27.545;
   1:L PR[91] R[100]mm/sec CNT100;
   1:  PR[91,1] = PR[90,1] + -32.598;
   1:  PR[91,2] = PR[90,2] + 5.722;
   1:  PR[91,3] = PR[90,3] + 27.550;
   1:L PR[91] R[100]mm/sec CNT100;
   1:  PR[91,1] = PR[90,1] + -32.792;
   1:  PR[91,2] = PR[90,2] + 5.114;
   1:  PR[91,3] = PR[90,3] + 27.554;
   1:L PR[91] R[100]mm/sec CNT100;
   1:  PR[91,1] = PR[90,1] + -32.937;
   1:  PR[91,2] = PR[90,2] + 4.593;
   1:  PR[91,3] = PR[90,3] + 27.558;
   1:L PR[91] R[100]mm/sec CNT100;
   1:  PR[91,1] = PR[90,1] + -33.082;
   1:  PR[91,2] = PR[90,2] + 3.993;
   1:  PR[91,3] = PR[90,3] + 27.562;
   1:L PR[91] R[100]mm/sec CNT100;
   1:  PR[91,1] = PR[90,1] + -33.201;
   1:  PR[91,2] = PR[90,2] + 3.400;
   1:  PR[91,3] = PR[90,3] + 27.567;
   1:L PR[91] R[100]mm/sec CNT100;
   1:  PR[91,1] = PR[90,1] + -33.295;
   1:  PR[91,2] = PR[90,2] + 2.807;
   1:  PR[91,3] = PR[90,3] + 27.572;
   1:L PR[91] R[100]mm/sec CNT100;
   1:  PR[91,1] = PR[90,1] + -33.363;
   1:  PR[91,2] = PR[90,2] + 2.248;
   1:  PR[91,3] = PR[90,3] + 27.576;
   1:L PR[91] R[100]mm/sec CNT100;
   1:  PR[91,1] = PR[90,1] + -33.414;
   1:  PR[91,2] = PR[90,2] + 1.641;
   1:  PR[91,3] = PR[90,3] + 27.580;
   1:L PR[91] R[100]mm/sec CNT100;
   1:  PR[91,1] = PR[90,1] + -33.443;
   1:  PR[91,2] = PR[90,2] + 1.056;
   1:  PR[91,3] = PR[90,3] + 27.585;
   1:L PR[91] R[100]mm/sec CNT100;
   1:  PR[91,1] = PR[90,1] + -33.454;
   1:  PR[91,2] = PR[90,2] + 0.428;
   1:  PR[91,3] = PR[90,3] + 27.589;
   1:L PR[91] R[100]mm/sec CNT100;
   1:  PR[91,1] = PR[90,1] + -33.443;
   1:  PR[91,2] = PR[90,2] + -0.201;
   1:  PR[91,3] = PR[90,3] + 27.594;
   1:L PR[91] R[100]mm/sec CNT100;
   1:  PR[91,1] = PR[90,1] + -33.414;
   1:  PR[91,2] = PR[90,2] + -0.786;
   1:  PR[91,3] = PR[90,3] + 27.599;
   1:L PR[91] R[100]mm/sec CNT100;
   1:  PR[91,1] = PR[90,1] + -33.363;
   1:  PR[91,2] = PR[90,2] + -1.393;
   1:  PR[91,3] = PR[90,3] + 27.603;
   1:L PR[91] R[100]mm/sec CNT100;
   1:  PR[91,1] = PR[90,1] + -33.289;
   1:  PR[91,2] = PR[90,2] + -1.995;
   1:  PR[91,3] = PR[90,3] + 27.608;
   1:L PR[91] R[100]mm/sec CNT100;
   1:  PR[91,1] = PR[90,1] + -33.201;
   1:  PR[91,2] = PR[90,2] + -2.544;
   1:  PR[91,3] = PR[90,3] + 27.612;
   1:L PR[91] R[100]mm/sec CNT100;
   1:  PR[91,1] = PR[90,1] + -33.082;
   1:  PR[91,2] = PR[90,2] + -3.138;
   1:  PR[91,3] = PR[90,3] + 27.616;
   1:L PR[91] R[100]mm/sec CNT100;
   1:  PR[91,1] = PR[90,1] + -32.937;
   1:  PR[91,2] = PR[90,2] + -3.737;
   1:  PR[91,3] = PR[90,3] + 27.621;
   1:L PR[91] R[100]mm/sec CNT100;
   1:  PR[91,1] = PR[90,1] + -32.792;
   1:  PR[91,2] = PR[90,2] + -4.259;
   1:  PR[91,3] = PR[90,3] + 27.625;
   1:L PR[91] R[100]mm/sec CNT100;
   1:  PR[91,1] = PR[90,1] + -32.598;
   1:  PR[91,2] = PR[90,2] + -4.866;
   1:  PR[91,3] = PR[90,3] + 27.629;
   1:L PR[91] R[100]mm/sec CNT100;
   1:  PR[91,1] = PR[90,1] + -32.372;
   1:  PR[91,2] = PR[90,2] + -5.490;
   1:  PR[91,3] = PR[90,3] + 27.634;
   1:L PR[91] R[100]mm/sec CNT100;
   1:  PR[91,1] = PR[90,1] + -32.173;
   1:  PR[91,2] = PR[90,2] + -5.989;
   1:  PR[91,3] = PR[90,3] + 27.639;
   1:L PR[91] R[100]mm/sec CNT100;
   1:  PR[91,1] = PR[90,1] + -31.894;
   1:  PR[91,2] = PR[90,2] + -6.624;
   1:  PR[91,3] = PR[90,3] + 27.643;
   1:L PR[91] R[100]mm/sec CNT100;
   1:  PR[91,1] = PR[90,1] + -31.584;
   1:  PR[91,2] = PR[90,2] + -7.262;
   1:  PR[91,3] = PR[90,3] + 27.648;
   1:L PR[91] R[100]mm/sec CNT100;
   1:  PR[91,1] = PR[90,1] + -31.001;
   1:  PR[91,2] = PR[90,2] + -8.322;
   1:  PR[91,3] = PR[90,3] + 27.654;
   1:L PR[91] R[100]mm/sec CNT100;
   1:  PR[91,1] = PR[90,1] + -30.617;
   1:  PR[91,2] = PR[90,2] + -8.939;
   1:  PR[91,3] = PR[90,3] + 27.663;
   1:L PR[91] R[100]mm/sec CNT100;
   1:  PR[91,1] = PR[90,1] + -30.186;
   1:  PR[91,2] = PR[90,2] + -9.568;
   1:  PR[91,3] = PR[90,3] + 27.668;
   1:L PR[91] R[100]mm/sec CNT100;
   1:  PR[91,1] = PR[90,1] + -29.957;
   1:  PR[91,2] = PR[90,2] + -9.886;
   1:  PR[91,3] = PR[90,3] + 27.674;
   1:L PR[91] R[100]mm/sec CNT100;
   1:  PR[91,1] = PR[90,1] + -29.488;
   1:  PR[91,2] = PR[90,2] + -10.487;
   1:  PR[91,3] = PR[90,3] + 27.677;
   1:L PR[91] R[100]mm/sec CNT100;
   1:  PR[91,1] = PR[90,1] + -28.755;
   1:  PR[91,2] = PR[90,2] + -11.329;
   1:  PR[91,3] = PR[90,3] + 27.683;
   1:L PR[91] R[100]mm/sec CNT100;
   1:  PR[91,1] = PR[90,1] + -28.000;
   1:  PR[91,2] = PR[90,2] + -12.096;
   1:  PR[91,3] = PR[90,3] + 27.691;
   1:L PR[91] R[100]mm/sec CNT100;
   1:  PR[91,1] = PR[90,1] + -27.399;
   1:  PR[91,2] = PR[90,2] + -12.648;
   1:  PR[91,3] = PR[90,3] + 27.699;
   1:L PR[91] R[100]mm/sec CNT100;
   1:  PR[91,1] = PR[90,1] + -26.587;
   1:  PR[91,2] = PR[90,2] + -13.320;
   1:  PR[91,3] = PR[90,3] + 27.705;
   1:L PR[91] R[100]mm/sec CNT100;
   1:  PR[91,1] = PR[90,1] + -25.889;
   1:  PR[91,2] = PR[90,2] + -13.842;
   1:  PR[91,3] = PR[90,3] + 27.713;
   1:L PR[91] R[100]mm/sec CNT100;
   1:  PR[91,1] = PR[90,1] + -25.126;
   1:  PR[91,2] = PR[90,2] + -14.358;
   1:  PR[91,3] = PR[90,3] + 27.720;
   1:L PR[91] R[100]mm/sec CNT100;
   1:  PR[91,1] = PR[90,1] + -24.251;
   1:  PR[91,2] = PR[90,2] + -14.889;
   1:  PR[91,3] = PR[90,3] + 27.726;
   1:L PR[91] R[100]mm/sec CNT100;
   1:  PR[91,1] = PR[90,1] + -23.389;
   1:  PR[91,2] = PR[90,2] + -15.354;
   1:  PR[91,3] = PR[90,3] + 27.734;
   1:L PR[91] R[100]mm/sec CNT100;
   1:  PR[91,1] = PR[90,1] + -22.503;
   1:  PR[91,2] = PR[90,2] + -15.779;
   1:  PR[91,3] = PR[90,3] + 27.741;
   1:L PR[91] R[100]mm/sec CNT100;
   1:  PR[91,1] = PR[90,1] + -21.593;
   1:  PR[91,2] = PR[90,2] + -16.162;
   1:  PR[91,3] = PR[90,3] + 27.749;
   1:L PR[91] R[100]mm/sec CNT100;
   1:  PR[91,1] = PR[90,1] + -20.663;
   1:  PR[91,2] = PR[90,2] + -16.501;
   1:  PR[91,3] = PR[90,3] + 27.756;
   1:L PR[91] R[100]mm/sec CNT100;
   1:  PR[91,1] = PR[90,1] + -19.714;
   1:  PR[91,2] = PR[90,2] + -16.794;
   1:  PR[91,3] = PR[90,3] + 27.764;
   1:L PR[91] R[100]mm/sec CNT100;
   1:  PR[91,1] = PR[90,1] + -18.749;
   1:  PR[91,2] = PR[90,2] + -17.039;
   1:  PR[91,3] = PR[90,3] + 27.771;
   1:L PR[91] R[100]mm/sec CNT100;
   1:  PR[91,1] = PR[90,1] + -17.770;
   1:  PR[91,2] = PR[90,2] + -17.238;
   1:  PR[91,3] = PR[90,3] + 27.778;
   1:L PR[91] R[100]mm/sec CNT100;
   1:  PR[91,1] = PR[90,1] + -16.780;
   1:  PR[91,2] = PR[90,2] + -17.389;
   1:  PR[91,3] = PR[90,3] + 27.786;
   1:L PR[91] R[100]mm/sec CNT100;
   1:  PR[91,1] = PR[90,1] + -16.401;
   1:  PR[91,2] = PR[90,2] + -17.428;
   1:  PR[91,3] = PR[90,3] + 27.793;
   1:L PR[91] R[100]mm/sec CNT100;
   1:  PR[91,1] = PR[90,1] + -15.783;
   1:  PR[91,2] = PR[90,2] + -17.490;
   1:  PR[91,3] = PR[90,3] + 27.796;
   1:L PR[91] R[100]mm/sec CNT100;
   1:  PR[91,1] = PR[90,1] + -14.780;
   1:  PR[91,2] = PR[90,2] + -17.543;
   1:  PR[91,3] = PR[90,3] + 27.801;
   1:L PR[91] R[100]mm/sec CNT100;
   1:  PR[91,1] = PR[90,1] + -13.774;
   1:  PR[91,2] = PR[90,2] + -17.546;
   1:  PR[91,3] = PR[90,3] + 27.808;
   1:L PR[91] R[100]mm/sec CNT100;
   1:  PR[91,1] = PR[90,1] + -12.769;
   1:  PR[91,2] = PR[90,2] + -17.498;
   1:  PR[91,3] = PR[90,3] + 27.816;
   1:L PR[91] R[100]mm/sec CNT100;
   1:  PR[91,1] = PR[90,1] + -11.749;
   1:  PR[91,2] = PR[90,2] + -17.399;
   1:  PR[91,3] = PR[90,3] + 27.824;
   1:L PR[91] R[100]mm/sec CNT100;
   1:  PR[91,1] = PR[90,1] + -10.805;
   1:  PR[91,2] = PR[90,2] + -17.261;
   1:  PR[91,3] = PR[90,3] + 27.831;
   1:L PR[91] R[100]mm/sec CNT100;
   1:  PR[91,1] = PR[90,1] + -9.732;
   1:  PR[91,2] = PR[90,2] + -17.049;
   1:  PR[91,3] = PR[90,3] + 27.838;
   1:L PR[91] R[100]mm/sec CNT100;
   1:  PR[91,1] = PR[90,1] + -8.735;
   1:  PR[91,2] = PR[90,2] + -16.796;
   1:  PR[91,3] = PR[90,3] + 27.847;
   1:L PR[91] R[100]mm/sec CNT100;
   1:  PR[91,1] = PR[90,1] + -7.756;
   1:  PR[91,2] = PR[90,2] + -16.492;
   1:  PR[91,3] = PR[90,3] + 27.854;
   1:L PR[91] R[100]mm/sec CNT100;
   1:  PR[91,1] = PR[90,1] + -6.795;
   1:  PR[91,2] = PR[90,2] + -16.138;
   1:  PR[91,3] = PR[90,3] + 27.862;
   1:L PR[91] R[100]mm/sec CNT100;
   1:  PR[91,1] = PR[90,1] + -6.232;
   1:  PR[91,2] = PR[90,2] + -15.903;
   1:  PR[91,3] = PR[90,3] + 27.870;
   1:L PR[91] R[100]mm/sec CNT100;
   1:  PR[91,1] = PR[90,1] + -5.867;
   1:  PR[91,2] = PR[90,2] + -15.741;
   1:  PR[91,3] = PR[90,3] + 27.874;
   1:L PR[91] R[100]mm/sec CNT100;
   1:  PR[91,1] = PR[90,1] + -4.955;
   1:  PR[91,2] = PR[90,2] + -15.293;
   1:  PR[91,3] = PR[90,3] + 27.877;
   1:L PR[91] R[100]mm/sec CNT100;
   1:  PR[91,1] = PR[90,1] + -4.076;
   1:  PR[91,2] = PR[90,2] + -14.803;
   1:  PR[91,3] = PR[90,3] + 27.885;
   1:L PR[91] R[100]mm/sec CNT100;
   1:  PR[91,1] = PR[90,1] + -3.225;
   1:  PR[91,2] = PR[90,2] + -14.269;
   1:  PR[91,3] = PR[90,3] + 27.892;
   1:L PR[91] R[100]mm/sec CNT100;
   1:  PR[91,1] = PR[90,1] + -2.931;
   1:  PR[91,2] = PR[90,2] + -14.068;
   1:  PR[91,3] = PR[90,3] + 27.900;
   1:L PR[91] R[100]mm/sec CNT100;
   1:  PR[91,1] = PR[90,1] + -2.415;
   1:  PR[91,2] = PR[90,2] + -13.699;
   1:  PR[91,3] = PR[90,3] + 27.902;
   1:L PR[91] R[100]mm/sec CNT100;
   1:  PR[91,1] = PR[90,1] + -1.942;
   1:  PR[91,2] = PR[90,2] + -13.332;
   1:  PR[91,3] = PR[90,3] + 27.907;
   1:L PR[91] R[100]mm/sec CNT100;
   1:  PR[91,1] = PR[90,1] + -1.555;
   1:  PR[91,2] = PR[90,2] + -13.069;
   1:  PR[91,3] = PR[90,3] + 27.912;
   1:L PR[91] R[100]mm/sec CNT100;
   1:  PR[91,1] = PR[90,1] + -1.107;
   1:  PR[91,2] = PR[90,2] + -12.866;
   1:  PR[91,3] = PR[90,3] + 27.915;
   1:L PR[91] R[100]mm/sec CNT100;
   1:  PR[91,1] = PR[90,1] + -0.782;
   1:  PR[91,2] = PR[90,2] + -12.776;
   1:  PR[91,3] = PR[90,3] + 27.919;
   1:L PR[91] R[100]mm/sec CNT100;
   1:  PR[91,1] = PR[90,1] + -0.621;
   1:  PR[91,2] = PR[90,2] + -12.737;
   1:  PR[91,3] = PR[90,3] + 27.921;
   1:L PR[91] R[100]mm/sec CNT100;
   1:  PR[91,1] = PR[90,1] + -0.137;
   1:  PR[91,2] = PR[90,2] + -12.692;
   1:  PR[91,3] = PR[90,3] + 27.923;
   1:L PR[91] R[100]mm/sec CNT100;
   1:  PR[91,1] = PR[90,1] + 0.357;
   1:  PR[91,2] = PR[90,2] + -12.732;
   1:  PR[91,3] = PR[90,3] + 27.926;
   1:L PR[91] R[100]mm/sec CNT100;
   1:  PR[91] = PR[90];
   1:  PR[91,1] = PR[90,1] + 0.930;
   1:  PR[91,2] = PR[90,2] + -13.461;
   1:  PR[91,3] = PR[90,3] + 29.260;
   1:L PR[91] R[100]mm/sec CNT100;
   1:  PR[91,1] = PR[90,1] + 1.381;
   1:  PR[91,2] = PR[90,2] + -13.679;
   1:  PR[91,3] = PR[90,3] + 27.934;
   1:L PR[91] R[100]mm/sec CNT100;
   1:  PR[91,1] = PR[90,1] + 2.303;
   1:  PR[91,2] = PR[90,2] + -14.325;
   1:  PR[91,3] = PR[90,3] + 27.938;
   1:L PR[91] R[100]mm/sec CNT100;
   1:  PR[91,1] = PR[90,1] + 3.119;
   1:  PR[91,2] = PR[90,2] + -14.844;
   1:  PR[91,3] = PR[90,3] + 27.946;
   1:L PR[91] R[100]mm/sec CNT100;
   1:  PR[91,1] = PR[90,1] + 3.973;
   1:  PR[91,2] = PR[90,2] + -15.330;
   1:  PR[91,3] = PR[90,3] + 27.953;
   1:L PR[91] R[100]mm/sec CNT100;
   1:  PR[91,1] = PR[90,1] + 4.867;
   1:  PR[91,2] = PR[90,2] + -15.779;
   1:  PR[91,3] = PR[90,3] + 27.961;
   1:L PR[91] R[100]mm/sec CNT100;
   1:  PR[91,1] = PR[90,1] + 5.783;
   1:  PR[91,2] = PR[90,2] + -16.182;
   1:  PR[91,3] = PR[90,3] + 27.968;
   1:L PR[91] R[100]mm/sec CNT100;
   1:  PR[91,1] = PR[90,1] + 6.721;
   1:  PR[91,2] = PR[90,2] + -16.540;
   1:  PR[91,3] = PR[90,3] + 27.976;
   1:L PR[91] R[100]mm/sec CNT100;
   1:  PR[91,1] = PR[90,1] + 7.402;
   1:  PR[91,2] = PR[90,2] + -16.765;
   1:  PR[91,3] = PR[90,3] + 27.984;
   1:L PR[91] R[100]mm/sec CNT100;
   1:  PR[91,1] = PR[90,1] + 8.647;
   1:  PR[91,2] = PR[90,2] + -17.113;
   1:  PR[91,3] = PR[90,3] + 27.989;
   1:L PR[91] R[100]mm/sec CNT100;
   1:  PR[91,1] = PR[90,1] + 9.626;
   1:  PR[91,2] = PR[90,2] + -17.325;
   1:  PR[91,3] = PR[90,3] + 27.999;
   1:L PR[91] R[100]mm/sec CNT100;
   1:  PR[91,1] = PR[90,1] + 10.616;
   1:  PR[91,2] = PR[90,2] + -17.489;
   1:  PR[91,3] = PR[90,3] + 28.006;
   1:L PR[91] R[100]mm/sec CNT100;
   1:  PR[91,1] = PR[90,1] + 11.615;
   1:  PR[91,2] = PR[90,2] + -17.603;
   1:  PR[91,3] = PR[90,3] + 28.014;
   1:L PR[91] R[100]mm/sec CNT100;
   1:  PR[91,1] = PR[90,1] + 11.992;
   1:  PR[91,2] = PR[90,2] + -17.630;
   1:  PR[91,3] = PR[90,3] + 28.022;
   1:L PR[91] R[100]mm/sec CNT100;
   1:  PR[91,1] = PR[90,1] + 12.612;
   1:  PR[91,2] = PR[90,2] + -17.667;
   1:  PR[91,3] = PR[90,3] + 28.024;
   1:L PR[91] R[100]mm/sec CNT100;
   1:  PR[91,1] = PR[90,1] + 13.615;
   1:  PR[91,2] = PR[90,2] + -17.682;
   1:  PR[91,3] = PR[90,3] + 28.029;
   1:L PR[91] R[100]mm/sec CNT100;
   1:  PR[91,1] = PR[90,1] + 14.615;
   1:  PR[91,2] = PR[90,2] + -17.647;
   1:  PR[91,3] = PR[90,3] + 28.037;
   1:L PR[91] R[100]mm/sec CNT100;
   1:  PR[91,1] = PR[90,1] + 15.609;
   1:  PR[91,2] = PR[90,2] + -17.564;
   1:  PR[91,3] = PR[90,3] + 28.044;
   1:L PR[91] R[100]mm/sec CNT100;
   1:  PR[91,1] = PR[90,1] + 16.613;
   1:  PR[91,2] = PR[90,2] + -17.429;
   1:  PR[91,3] = PR[90,3] + 28.052;
   1:L PR[91] R[100]mm/sec CNT100;
   1:  PR[91,1] = PR[90,1] + 17.534;
   1:  PR[91,2] = PR[90,2] + -17.262;
   1:  PR[91,3] = PR[90,3] + 28.060;
   1:L PR[91] R[100]mm/sec CNT100;
   1:  PR[91,1] = PR[90,1] + 18.452;
   1:  PR[91,2] = PR[90,2] + -17.051;
   1:  PR[91,3] = PR[90,3] + 28.067;
   1:L PR[91] R[100]mm/sec CNT100;
   1:  PR[91,1] = PR[90,1] + 19.360;
   1:  PR[91,2] = PR[90,2] + -16.798;
   1:  PR[91,3] = PR[90,3] + 28.074;
   1:L PR[91] R[100]mm/sec CNT100;
   1:  PR[91,1] = PR[90,1] + 20.256;
   1:  PR[91,2] = PR[90,2] + -16.503;
   1:  PR[91,3] = PR[90,3] + 28.081;
   1:L PR[91] R[100]mm/sec CNT100;
   1:  PR[91,1] = PR[90,1] + 21.138;
   1:  PR[91,2] = PR[90,2] + -16.166;
   1:  PR[91,3] = PR[90,3] + 28.088;
   1:L PR[91] R[100]mm/sec CNT100;
   1:  PR[91,1] = PR[90,1] + 22.003;
   1:  PR[91,2] = PR[90,2] + -15.789;
   1:  PR[91,3] = PR[90,3] + 28.095;
   1:L PR[91] R[100]mm/sec CNT100;
   1:  PR[91,1] = PR[90,1] + 22.849;
   1:  PR[91,2] = PR[90,2] + -15.372;
   1:  PR[91,3] = PR[90,3] + 28.102;
   1:L PR[91] R[100]mm/sec CNT100;
   1:  PR[91,1] = PR[90,1] + 23.674;
   1:  PR[91,2] = PR[90,2] + -14.916;
   1:  PR[91,3] = PR[90,3] + 28.110;
   1:L PR[91] R[100]mm/sec CNT100;
   1:  PR[91,1] = PR[90,1] + 24.475;
   1:  PR[91,2] = PR[90,2] + -14.421;
   1:  PR[91,3] = PR[90,3] + 28.117;
   1:L PR[91] R[100]mm/sec CNT100;
   1:  PR[91,1] = PR[90,1] + 25.251;
   1:  PR[91,2] = PR[90,2] + -13.889;
   1:  PR[91,3] = PR[90,3] + 28.124;
   1:L PR[91] R[100]mm/sec CNT100;
   1:  PR[91,1] = PR[90,1] + 25.999;
   1:  PR[91,2] = PR[90,2] + -13.319;
   1:  PR[91,3] = PR[90,3] + 28.131;
   1:L PR[91] R[100]mm/sec CNT100;
   1:  PR[91,1] = PR[90,1] + 26.718;
   1:  PR[91,2] = PR[90,2] + -12.714;
   1:  PR[91,3] = PR[90,3] + 28.138;
   1:L PR[91] R[100]mm/sec CNT100;
   1:  PR[91,1] = PR[90,1] + 27.341;
   1:  PR[91,2] = PR[90,2] + -12.134;
   1:  PR[91,3] = PR[90,3] + 28.145;
   1:L PR[91] R[100]mm/sec CNT100;
   1:  PR[91,1] = PR[90,1] + 28.058;
   1:  PR[91,2] = PR[90,2] + -11.396;
   1:  PR[91,3] = PR[90,3] + 28.152;
   1:L PR[91] R[100]mm/sec CNT100;
   1:  PR[91,1] = PR[90,1] + 28.686;
   1:  PR[91,2] = PR[90,2] + -10.675;
   1:  PR[91,3] = PR[90,3] + 28.159;
   1:L PR[91] R[100]mm/sec CNT100;
   1:  PR[91,1] = PR[90,1] + 29.266;
   1:  PR[91,2] = PR[90,2] + -9.937;
   1:  PR[91,3] = PR[90,3] + 28.167;
   1:L PR[91] R[100]mm/sec CNT100;
   1:  PR[91,1] = PR[90,1] + 29.786;
   1:  PR[91,2] = PR[90,2] + -9.198;
   1:  PR[91,3] = PR[90,3] + 28.174;
   1:L PR[91] R[100]mm/sec CNT100;
   1:  PR[91,1] = PR[90,1] + 30.316;
   1:  PR[91,2] = PR[90,2] + -8.360;
   1:  PR[91,3] = PR[90,3] + 28.181;
   1:L PR[91] R[100]mm/sec CNT100;
   1:  PR[91,1] = PR[90,1] + 30.742;
   1:  PR[91,2] = PR[90,2] + -7.604;
   1:  PR[91,3] = PR[90,3] + 28.188;
   1:L PR[91] R[100]mm/sec CNT100;
   1:  PR[91,1] = PR[90,1] + 31.198;
   1:  PR[91,2] = PR[90,2] + -6.696;
   1:  PR[91,3] = PR[90,3] + 28.195;
   1:L PR[91] R[100]mm/sec CNT100;
   1:  PR[91,1] = PR[90,1] + 31.532;
   1:  PR[91,2] = PR[90,2] + -5.936;
   1:  PR[91,3] = PR[90,3] + 28.202;
   1:L PR[91] R[100]mm/sec CNT100;
   1:  PR[91,1] = PR[90,1] + 31.892;
   1:  PR[91,2] = PR[90,2] + -4.989;
   1:  PR[91,3] = PR[90,3] + 28.209;
   1:L PR[91] R[100]mm/sec CNT100;
   1:  PR[91,1] = PR[90,1] + 32.131;
   1:  PR[91,2] = PR[90,2] + -4.240;
   1:  PR[91,3] = PR[90,3] + 28.216;
   1:L PR[91] R[100]mm/sec CNT100;
   1:  PR[91,1] = PR[90,1] + 32.383;
   1:  PR[91,2] = PR[90,2] + -3.268;
   1:  PR[91,3] = PR[90,3] + 28.222;
   1:L PR[91] R[100]mm/sec CNT100;
   1:  PR[91,1] = PR[90,1] + 32.533;
   1:  PR[91,2] = PR[90,2] + -2.509;
   1:  PR[91,3] = PR[90,3] + 28.230;
   1:L PR[91] R[100]mm/sec CNT100;
   1:  PR[91,1] = PR[90,1] + 32.646;
   1:  PR[91,2] = PR[90,2] + -1.733;
   1:  PR[91,3] = PR[90,3] + 28.236;
   1:L PR[91] R[100]mm/sec CNT100;
   1:  PR[91,1] = PR[90,1] + 32.700;
   1:  PR[91,2] = PR[90,2] + -1.225;
   1:  PR[91,3] = PR[90,3] + 28.242;
   1:L PR[91] R[100]mm/sec CNT100;
   1:  PR[91,1] = PR[90,1] + 32.758;
   1:  PR[91,2] = PR[90,2] + -0.409;
   1:  PR[91,3] = PR[90,3] + 28.246;
   1:L PR[91] R[100]mm/sec CNT100;
   1:  PR[91,1] = PR[90,1] + 32.777;
   1:  PR[91,2] = PR[90,2] + 0.425;
   1:  PR[91,3] = PR[90,3] + 28.252;
   1:L PR[91] R[100]mm/sec CNT100;
   1:  PR[91,1] = PR[90,1] + 32.744;
   1:  PR[91,2] = PR[90,2] + 1.537;
   1:  PR[91,3] = PR[90,3] + 28.258;
   1:L PR[91] R[100]mm/sec CNT100;
   1:  PR[91,1] = PR[90,1] + 32.678;
   1:  PR[91,2] = PR[90,2] + 2.336;
   1:  PR[91,3] = PR[90,3] + 28.267;
   1:L PR[91] R[100]mm/sec CNT100;
   1:  PR[91,1] = PR[90,1] + 32.533;
   1:  PR[91,2] = PR[90,2] + 3.366;
   1:  PR[91,3] = PR[90,3] + 28.273;
   1:L PR[91] R[100]mm/sec CNT100;
   1:  PR[91,1] = PR[90,1] + 32.383;
   1:  PR[91,2] = PR[90,2] + 4.123;
   1:  PR[91,3] = PR[90,3] + 28.280;
   1:L PR[91] R[100]mm/sec CNT100;
   1:  PR[91,1] = PR[90,1] + 32.131;
   1:  PR[91,2] = PR[90,2] + 5.095;
   1:  PR[91,3] = PR[90,3] + 28.286;
   1:L PR[91] R[100]mm/sec CNT100;
   1:  PR[91,1] = PR[90,1] + 31.892;
   1:  PR[91,2] = PR[90,2] + 5.844;
   1:  PR[91,3] = PR[90,3] + 28.294;
   1:L PR[91] R[100]mm/sec CNT100;
   1:  PR[91,1] = PR[90,1] + 31.532;
   1:  PR[91,2] = PR[90,2] + 6.792;
   1:  PR[91,3] = PR[90,3] + 28.300;
   1:L PR[91] R[100]mm/sec CNT100;
   1:  PR[91,1] = PR[90,1] + 31.197;
   1:  PR[91,2] = PR[90,2] + 7.552;
   1:  PR[91,3] = PR[90,3] + 28.308;
   1:L PR[91] R[100]mm/sec CNT100;
   1:  PR[91,1] = PR[90,1] + 30.742;
   1:  PR[91,2] = PR[90,2] + 8.460;
   1:  PR[91,3] = PR[90,3] + 28.314;
   1:L PR[91] R[100]mm/sec CNT100;
   1:  PR[91,1] = PR[90,1] + 30.316;
   1:  PR[91,2] = PR[90,2] + 9.216;
   1:  PR[91,3] = PR[90,3] + 28.322;
   1:L PR[91] R[100]mm/sec CNT100;
   1:  PR[91,1] = PR[90,1] + 29.786;
   1:  PR[91,2] = PR[90,2] + 10.054;
   1:  PR[91,3] = PR[90,3] + 28.328;
   1:L PR[91] R[100]mm/sec CNT100;
   1:  PR[91,1] = PR[90,1] + 29.265;
   1:  PR[91,2] = PR[90,2] + 10.792;
   1:  PR[91,3] = PR[90,3] + 28.336;
   1:L PR[91] R[100]mm/sec CNT100;
   1:  PR[91,1] = PR[90,1] + 28.673;
   1:  PR[91,2] = PR[90,2] + 11.546;
   1:  PR[91,3] = PR[90,3] + 28.342;
   1:L PR[91] R[100]mm/sec CNT100;
   1:  PR[91,1] = PR[90,1] + 28.040;
   1:  PR[91,2] = PR[90,2] + 12.271;
   1:  PR[91,3] = PR[90,3] + 28.350;
   1:L PR[91] R[100]mm/sec CNT100;
   1:  PR[91,1] = PR[90,1] + 27.341;
   1:  PR[91,2] = PR[90,2] + 12.989;
   1:  PR[91,3] = PR[90,3] + 28.357;
   1:L PR[91] R[100]mm/sec CNT100;
   1:  PR[91,1] = PR[90,1] + 26.718;
   1:  PR[91,2] = PR[90,2] + 13.569;
   1:  PR[91,3] = PR[90,3] + 28.365;
   1:L PR[91] R[100]mm/sec CNT100;
   1:  PR[91,1] = PR[90,1] + 25.999;
   1:  PR[91,2] = PR[90,2] + 14.175;
   1:  PR[91,3] = PR[90,3] + 28.371;
   1:L PR[91] R[100]mm/sec CNT100;
   1:  PR[91,1] = PR[90,1] + 25.250;
   1:  PR[91,2] = PR[90,2] + 14.744;
   1:  PR[91,3] = PR[90,3] + 28.378;
   1:L PR[91] R[100]mm/sec CNT100;
   1:  PR[91,1] = PR[90,1] + 24.475;
   1:  PR[91,2] = PR[90,2] + 15.276;
   1:  PR[91,3] = PR[90,3] + 28.385;
   1:L PR[91] R[100]mm/sec CNT100;
   1:  PR[91,1] = PR[90,1] + 23.673;
   1:  PR[91,2] = PR[90,2] + 15.771;
   1:  PR[91,3] = PR[90,3] + 28.392;
   1:L PR[91] R[100]mm/sec CNT100;
   1:  PR[91,1] = PR[90,1] + 22.849;
   1:  PR[91,2] = PR[90,2] + 16.227;
   1:  PR[91,3] = PR[90,3] + 28.400;
   1:L PR[91] R[100]mm/sec CNT100;
   1:  PR[91,1] = PR[90,1] + 22.003;
   1:  PR[91,2] = PR[90,2] + 16.644;
   1:  PR[91,3] = PR[90,3] + 28.407;
   1:L PR[91] R[100]mm/sec CNT100;
   1:  PR[91,1] = PR[90,1] + 21.137;
   1:  PR[91,2] = PR[90,2] + 17.021;
   1:  PR[91,3] = PR[90,3] + 28.414;
   1:L PR[91] R[100]mm/sec CNT100;
   1:  PR[91,1] = PR[90,1] + 20.256;
   1:  PR[91,2] = PR[90,2] + 17.358;
   1:  PR[91,3] = PR[90,3] + 28.421;
   1:L PR[91] R[100]mm/sec CNT100;
   1:  PR[91,1] = PR[90,1] + 19.360;
   1:  PR[91,2] = PR[90,2] + 17.653;
   1:  PR[91,3] = PR[90,3] + 28.428;
   1:L PR[91] R[100]mm/sec CNT100;
   1:  PR[91,1] = PR[90,1] + 18.452;
   1:  PR[91,2] = PR[90,2] + 17.906;
   1:  PR[91,3] = PR[90,3] + 28.435;
   1:L PR[91] R[100]mm/sec CNT100;
   1:  PR[91,1] = PR[90,1] + 17.534;
   1:  PR[91,2] = PR[90,2] + 18.117;
   1:  PR[91,3] = PR[90,3] + 28.442;
   1:L PR[91] R[100]mm/sec CNT100;
   1:  PR[91,1] = PR[90,1] + 16.597;
   1:  PR[91,2] = PR[90,2] + 18.287;
   1:  PR[91,3] = PR[90,3] + 28.450;
   1:L PR[91] R[100]mm/sec CNT100;
   1:  PR[91,1] = PR[90,1] + 15.610;
   1:  PR[91,2] = PR[90,2] + 18.419;
   1:  PR[91,3] = PR[90,3] + 28.457;
   1:L PR[91] R[100]mm/sec CNT100;
   1:  PR[91,1] = PR[90,1] + 14.615;
   1:  PR[91,2] = PR[90,2] + 18.502;
   1:  PR[91,3] = PR[90,3] + 28.464;
   1:L PR[91] R[100]mm/sec CNT100;
   1:  PR[91,1] = PR[90,1] + 13.615;
   1:  PR[91,2] = PR[90,2] + 18.537;
   1:  PR[91,3] = PR[90,3] + 28.472;
   1:L PR[91] R[100]mm/sec CNT100;
   1:  PR[91,1] = PR[90,1] + 12.612;
   1:  PR[91,2] = PR[90,2] + 18.522;
   1:  PR[91,3] = PR[90,3] + 28.479;
   1:L PR[91] R[100]mm/sec CNT100;
   1:  PR[91,1] = PR[90,1] + 11.992;
   1:  PR[91,2] = PR[90,2] + 18.485;
   1:  PR[91,3] = PR[90,3] + 28.487;
   1:L PR[91] R[100]mm/sec CNT100;
   1:  PR[91,1] = PR[90,1] + 11.615;
   1:  PR[91,2] = PR[90,2] + 18.458;
   1:  PR[91,3] = PR[90,3] + 28.492;
   1:L PR[91] R[100]mm/sec CNT100;
   1:  PR[91,1] = PR[90,1] + 10.616;
   1:  PR[91,2] = PR[90,2] + 18.344;
   1:  PR[91,3] = PR[90,3] + 28.495;
   1:L PR[91] R[100]mm/sec CNT100;
   1:  PR[91,1] = PR[90,1] + 9.625;
   1:  PR[91,2] = PR[90,2] + 18.180;
   1:  PR[91,3] = PR[90,3] + 28.502;
   1:L PR[91] R[100]mm/sec CNT100;
   1:  PR[91,1] = PR[90,1] + 8.646;
   1:  PR[91,2] = PR[90,2] + 17.968;
   1:  PR[91,3] = PR[90,3] + 28.510;
   1:L PR[91] R[100]mm/sec CNT100;
   1:  PR[91,1] = PR[90,1] + 7.402;
   1:  PR[91,2] = PR[90,2] + 17.620;
   1:  PR[91,3] = PR[90,3] + 28.517;
   1:L PR[91] R[100]mm/sec CNT100;
   1:  PR[91,1] = PR[90,1] + 6.720;
   1:  PR[91,2] = PR[90,2] + 17.395;
   1:  PR[91,3] = PR[90,3] + 28.527;
   1:L PR[91] R[100]mm/sec CNT100;
   1:  PR[91,1] = PR[90,1] + 5.782;
   1:  PR[91,2] = PR[90,2] + 17.037;
   1:  PR[91,3] = PR[90,3] + 28.533;
   1:L PR[91] R[100]mm/sec CNT100;
   1:  PR[91,1] = PR[90,1] + 4.866;
   1:  PR[91,2] = PR[90,2] + 16.634;
   1:  PR[91,3] = PR[90,3] + 28.540;
   1:L PR[91] R[100]mm/sec CNT100;
   1:  PR[91,1] = PR[90,1] + 3.973;
   1:  PR[91,2] = PR[90,2] + 16.184;
   1:  PR[91,3] = PR[90,3] + 28.548;
   1:L PR[91] R[100]mm/sec CNT100;
   1:  PR[91,1] = PR[90,1] + 3.102;
   1:  PR[91,2] = PR[90,2] + 15.689;
   1:  PR[91,3] = PR[90,3] + 28.555;
   1:L PR[91] R[100]mm/sec CNT100;
   1:  PR[91,1] = PR[90,1] + 2.291;
   1:  PR[91,2] = PR[90,2] + 15.172;
   1:  PR[91,3] = PR[90,3] + 28.563;
   1:L PR[91] R[100]mm/sec CNT100;
   1:  PR[91,1] = PR[90,1] + 1.381;
   1:  PR[91,2] = PR[90,2] + 14.534;
   1:  PR[91,3] = PR[90,3] + 28.570;
   1:L PR[91] R[100]mm/sec CNT100;
   1:  PR[91,1] = PR[90,1] + 0.930;
   1:  PR[91,2] = PR[90,2] + 14.316;
   1:  PR[91,3] = PR[90,3] + 28.579;
   1:L PR[91] R[100]mm/sec CNT100;
   1:  PR[91,1] = PR[90,1] + 0.453;
   1:  PR[91,2] = PR[90,2] + 14.180;
   1:  PR[91,3] = PR[90,3] + 28.583;
   1:L PR[91] R[100]mm/sec CNT100;
   1:  PR[91,1] = PR[90,1] + -0.039;
   1:  PR[91,2] = PR[90,2] + 14.121;
   1:  PR[91,3] = PR[90,3] + 28.586;
   1:L PR[91] R[100]mm/sec CNT100;
   1:  PR[91,1] = PR[90,1] + -0.532;
   1:  PR[91,2] = PR[90,2] + 14.152;
   1:  PR[91,3] = PR[90,3] + 28.590;
   1:L PR[91] R[100]mm/sec CNT100;
   1:  PR[91,1] = PR[90,1] + -1.010;
   1:  PR[91,2] = PR[90,2] + 14.261;
   1:  PR[91,3] = PR[90,3] + 28.594;
   1:L PR[91] R[100]mm/sec CNT100;
   1:  PR[91,1] = PR[90,1] + -1.466;
   1:  PR[91,2] = PR[90,2] + 14.449;
   1:  PR[91,3] = PR[90,3] + 28.597;
   1:L PR[91] R[100]mm/sec CNT100;
   1:  PR[91,1] = PR[90,1] + -1.859;
   1:  PR[91,2] = PR[90,2] + 14.693;
   1:  PR[91,3] = PR[90,3] + 28.601;
   1:L PR[91] R[100]mm/sec CNT100;
   1:  PR[91,1] = PR[90,1] + -2.534;
   1:  PR[91,2] = PR[90,2] + 15.172;
   1:  PR[91,3] = PR[90,3] + 28.605;
   1:L PR[91] R[100]mm/sec CNT100;
   1:  PR[91,1] = PR[90,1] + -3.360;
   1:  PR[91,2] = PR[90,2] + 15.698;
   1:  PR[91,3] = PR[90,3] + 28.611;
   1:L PR[91] R[100]mm/sec CNT100;
   1:  PR[91,1] = PR[90,1] + -4.218;
   1:  PR[91,2] = PR[90,2] + 16.186;
   1:  PR[91,3] = PR[90,3] + 28.618;
   1:L PR[91] R[100]mm/sec CNT100;
   1:  PR[91,1] = PR[90,1] + -5.120;
   1:  PR[91,2] = PR[90,2] + 16.640;
   1:  PR[91,3] = PR[90,3] + 28.626;
   1:L PR[91] R[100]mm/sec CNT100;
   1:  PR[91,1] = PR[90,1] + -6.048;
   1:  PR[91,2] = PR[90,2] + 17.049;
   1:  PR[91,3] = PR[90,3] + 28.634;
   1:L PR[91] R[100]mm/sec CNT100;
   1:  PR[91,1] = PR[90,1] + -7.002;
   1:  PR[91,2] = PR[90,2] + 17.411;
   1:  PR[91,3] = PR[90,3] + 28.641;
   1:L PR[91] R[100]mm/sec CNT100;
   1:  PR[91,1] = PR[90,1] + -7.689;
   1:  PR[91,2] = PR[90,2] + 17.638;
   1:  PR[91,3] = PR[90,3] + 28.649;
   1:L PR[91] R[100]mm/sec CNT100;
   1:  PR[91,1] = PR[90,1] + -8.611;
   1:  PR[91,2] = PR[90,2] + 17.900;
   1:  PR[91,3] = PR[90,3] + 28.654;
   1:L PR[91] R[100]mm/sec CNT100;
   1:  PR[91,1] = PR[90,1] + -9.548;
   1:  PR[91,2] = PR[90,2] + 18.117;
   1:  PR[91,3] = PR[90,3] + 28.662;
   1:L PR[91] R[100]mm/sec CNT100;
   1:  PR[91,1] = PR[90,1] + -9.968;
   1:  PR[91,2] = PR[90,2] + 18.200;
   1:  PR[91,3] = PR[90,3] + 28.669;
   1:L PR[91] R[100]mm/sec CNT100;
   1:  PR[91,1] = PR[90,1] + -10.994;
   1:  PR[91,2] = PR[90,2] + 18.362;
   1:  PR[91,3] = PR[90,3] + 28.672;
   1:L PR[91] R[100]mm/sec CNT100;
   1:  PR[91,1] = PR[90,1] + -12.024;
   1:  PR[91,2] = PR[90,2] + 18.471;
   1:  PR[91,3] = PR[90,3] + 28.680;
   1:L PR[91] R[100]mm/sec CNT100;
   1:  PR[91,1] = PR[90,1] + -13.369;
   1:  PR[91,2] = PR[90,2] + 18.535;
   1:  PR[91,3] = PR[90,3] + 28.688;
   1:L PR[91] R[100]mm/sec CNT100;
   1:  PR[91,1] = PR[90,1] + -14.333;
   1:  PR[91,2] = PR[90,2] + 18.525;
   1:  PR[91,3] = PR[90,3] + 28.698;
   1:L PR[91] R[100]mm/sec CNT100;
   1:  PR[91,1] = PR[90,1] + -15.151;
   1:  PR[91,2] = PR[90,2] + 18.481;
   1:  PR[91,3] = PR[90,3] + 28.705;
   1:L PR[91] R[100]mm/sec CNT100;
   1:  PR[91,1] = PR[90,1] + -16.195;
   1:  PR[91,2] = PR[90,2] + 18.377;
   1:  PR[91,3] = PR[90,3] + 28.712;
   1:L PR[91] R[100]mm/sec CNT100;
   1:  PR[91,1] = PR[90,1] + -17.225;
   1:  PR[91,2] = PR[90,2] + 18.221;
   1:  PR[91,3] = PR[90,3] + 28.720;
   1:L PR[91] R[100]mm/sec CNT100;
   1:  PR[91,1] = PR[90,1] + -18.211;
   1:  PR[91,2] = PR[90,2] + 18.023;
   1:  PR[91,3] = PR[90,3] + 28.727;
   1:L PR[91] R[100]mm/sec CNT100;
   1:  PR[91,1] = PR[90,1] + -19.183;
   1:  PR[91,2] = PR[90,2] + 17.777;
   1:  PR[91,3] = PR[90,3] + 28.735;
   1:L PR[91] R[100]mm/sec CNT100;
   1:  PR[91,1] = PR[90,1] + -20.138;
   1:  PR[91,2] = PR[90,2] + 17.484;
   1:  PR[91,3] = PR[90,3] + 28.743;
   1:L PR[91] R[100]mm/sec CNT100;
   1:  PR[91,1] = PR[90,1] + -21.075;
   1:  PR[91,2] = PR[90,2] + 17.145;
   1:  PR[91,3] = PR[90,3] + 28.750;
   1:L PR[91] R[100]mm/sec CNT100;
   1:  PR[91,1] = PR[90,1] + -21.991;
   1:  PR[91,2] = PR[90,2] + 16.760;
   1:  PR[91,3] = PR[90,3] + 28.758;
   1:L PR[91] R[100]mm/sec CNT100;
   1:  PR[91,1] = PR[90,1] + -22.884;
   1:  PR[91,2] = PR[90,2] + 16.333;
   1:  PR[91,3] = PR[90,3] + 28.765;
   1:L PR[91] R[100]mm/sec CNT100;
   1:  PR[91,1] = PR[90,1] + -23.751;
   1:  PR[91,2] = PR[90,2] + 15.863;
   1:  PR[91,3] = PR[90,3] + 28.773;
   1:L PR[91] R[100]mm/sec CNT100;
   1:  PR[91,1] = PR[90,1] + -24.589;
   1:  PR[91,2] = PR[90,2] + 15.354;
   1:  PR[91,3] = PR[90,3] + 28.780;
   1:L PR[91] R[100]mm/sec CNT100;
   1:  PR[91,1] = PR[90,1] + -25.398;
   1:  PR[91,2] = PR[90,2] + 14.807;
   1:  PR[91,3] = PR[90,3] + 28.788;
   1:L PR[91] R[100]mm/sec CNT100;
   1:  PR[91,1] = PR[90,1] + -26.174;
   1:  PR[91,2] = PR[90,2] + 14.223;
   1:  PR[91,3] = PR[90,3] + 28.795;
   1:L PR[91] R[100]mm/sec CNT100;
   1:  PR[91,1] = PR[90,1] + -26.916;
   1:  PR[91,2] = PR[90,2] + 13.603;
   1:  PR[91,3] = PR[90,3] + 28.802;
   1:L PR[91] R[100]mm/sec CNT100;
   1:  PR[91,1] = PR[90,1] + -27.621;
   1:  PR[91,2] = PR[90,2] + 12.949;
   1:  PR[91,3] = PR[90,3] + 28.810;
   1:L PR[91] R[100]mm/sec CNT100;
   1:  PR[91,1] = PR[90,1] + -28.289;
   1:  PR[91,2] = PR[90,2] + 12.263;
   1:  PR[91,3] = PR[90,3] + 28.817;
   1:L PR[91] R[100]mm/sec CNT100;
   1:  PR[91,1] = PR[90,1] + -28.924;
   1:  PR[91,2] = PR[90,2] + 11.537;
   1:  PR[91,3] = PR[90,3] + 28.824;
   1:L PR[91] R[100]mm/sec CNT100;
   1:  PR[91,1] = PR[90,1] + -29.505;
   1:  PR[91,2] = PR[90,2] + 10.800;
   1:  PR[91,3] = PR[90,3] + 28.832;
   1:L PR[91] R[100]mm/sec CNT100;
   1:  PR[91,1] = PR[90,1] + -30.076;
   1:  PR[91,2] = PR[90,2] + 9.987;
   1:  PR[91,3] = PR[90,3] + 28.839;
   1:L PR[91] R[100]mm/sec CNT100;
   1:  PR[91,1] = PR[90,1] + -30.555;
   1:  PR[91,2] = PR[90,2] + 9.223;
   1:  PR[91,3] = PR[90,3] + 28.846;
   1:L PR[91] R[100]mm/sec CNT100;
   1:  PR[91,1] = PR[90,1] + -30.982;
   1:  PR[91,2] = PR[90,2] + 8.462;
   1:  PR[91,3] = PR[90,3] + 28.853;
   1:L PR[91] R[100]mm/sec CNT100;
   1:  PR[91,1] = PR[90,1] + -31.438;
   1:  PR[91,2] = PR[90,2] + 7.545;
   1:  PR[91,3] = PR[90,3] + 28.860;
   1:L PR[91] R[100]mm/sec CNT100;
   1:  PR[91,1] = PR[90,1] + -31.773;
   1:  PR[91,2] = PR[90,2] + 6.775;
   1:  PR[91,3] = PR[90,3] + 28.867;
   1:L PR[91] R[100]mm/sec CNT100;
   1:  PR[91,1] = PR[90,1] + -32.134;
   1:  PR[91,2] = PR[90,2] + 5.817;
   1:  PR[91,3] = PR[90,3] + 28.874;
   1:L PR[91] R[100]mm/sec CNT100;
   1:  PR[91,1] = PR[90,1] + -32.436;
   1:  PR[91,2] = PR[90,2] + 4.840;
   1:  PR[91,3] = PR[90,3] + 28.882;
   1:L PR[91] R[100]mm/sec CNT100;
   1:  PR[91,1] = PR[90,1] + -32.627;
   1:  PR[91,2] = PR[90,2] + 4.081;
   1:  PR[91,3] = PR[90,3] + 28.889;
   1:L PR[91] R[100]mm/sec CNT100;
   1:  PR[91,1] = PR[90,1] + -32.777;
   1:  PR[91,2] = PR[90,2] + 3.323;
   1:  PR[91,3] = PR[90,3] + 28.895;
   1:L PR[91] R[100]mm/sec CNT100;
   1:  PR[91,1] = PR[90,1] + -32.919;
   1:  PR[91,2] = PR[90,2] + 2.304;
   1:  PR[91,3] = PR[90,3] + 28.901;
   1:L PR[91] R[100]mm/sec CNT100;
   1:  PR[91,1] = PR[90,1] + -32.984;
   1:  PR[91,2] = PR[90,2] + 1.515;
   1:  PR[91,3] = PR[90,3] + 28.909;
   1:L PR[91] R[100]mm/sec CNT100;
   1:  PR[91,1] = PR[90,1] + -33.015;
   1:  PR[91,2] = PR[90,2] + 0.424;
   1:  PR[91,3] = PR[90,3] + 28.915;
   1:L PR[91] R[100]mm/sec CNT100;
   1:  PR[91,1] = PR[90,1] + -33.011;
   1:  PR[91,2] = PR[90,2] + 0.166;
   1:  PR[91,3] = PR[90,3] + 28.923;
   1:L PR[91] R[100]mm/sec CNT100;
   1:  PR[91,1] = PR[90,1] + -32.984;
   1:  PR[91,2] = PR[90,2] + -0.658;
   1:  PR[91,3] = PR[90,3] + 28.925;
   1:L PR[91] R[100]mm/sec CNT100;
   1:  PR[91,1] = PR[90,1] + -32.919;
   1:  PR[91,2] = PR[90,2] + -1.449;
   1:  PR[91,3] = PR[90,3] + 28.931;
   1:L PR[91] R[100]mm/sec CNT100;
   1:  PR[91,1] = PR[90,1] + -32.777;
   1:  PR[91,2] = PR[90,2] + -2.468;
   1:  PR[91,3] = PR[90,3] + 28.937;
   1:L PR[91] R[100]mm/sec CNT100;
   1:  PR[91,1] = PR[90,1] + -32.627;
   1:  PR[91,2] = PR[90,2] + -3.226;
   1:  PR[91,3] = PR[90,3] + 28.945;
   1:L PR[91] R[100]mm/sec CNT100;
   1:  PR[91,1] = PR[90,1] + -32.436;
   1:  PR[91,2] = PR[90,2] + -3.985;
   1:  PR[91,3] = PR[90,3] + 28.951;
   1:L PR[91] R[100]mm/sec CNT100;
   1:  PR[91,1] = PR[90,1] + -32.134;
   1:  PR[91,2] = PR[90,2] + -4.961;
   1:  PR[91,3] = PR[90,3] + 28.957;
   1:L PR[91] R[100]mm/sec CNT100;
   1:  PR[91,1] = PR[90,1] + -31.773;
   1:  PR[91,2] = PR[90,2] + -5.920;
   1:  PR[91,3] = PR[90,3] + 28.965;
   1:L PR[91] R[100]mm/sec CNT100;
   1:  PR[91,1] = PR[90,1] + -31.438;
   1:  PR[91,2] = PR[90,2] + -6.690;
   1:  PR[91,3] = PR[90,3] + 28.972;
   1:L PR[91] R[100]mm/sec CNT100;
   1:  PR[91,1] = PR[90,1] + -30.982;
   1:  PR[91,2] = PR[90,2] + -7.607;
   1:  PR[91,3] = PR[90,3] + 28.979;
   1:L PR[91] R[100]mm/sec CNT100;
   1:  PR[91,1] = PR[90,1] + -30.556;
   1:  PR[91,2] = PR[90,2] + -8.367;
   1:  PR[91,3] = PR[90,3] + 28.987;
   1:L PR[91] R[100]mm/sec CNT100;
   1:  PR[91,1] = PR[90,1] + -30.076;
   1:  PR[91,2] = PR[90,2] + -9.131;
   1:  PR[91,3] = PR[90,3] + 28.993;
   1:L PR[91] R[100]mm/sec CNT100;
   1:  PR[91,1] = PR[90,1] + -29.505;
   1:  PR[91,2] = PR[90,2] + -9.945;
   1:  PR[91,3] = PR[90,3] + 29.000;
   1:L PR[91] R[100]mm/sec CNT100;
   1:  PR[91,1] = PR[90,1] + -28.912;
   1:  PR[91,2] = PR[90,2] + -10.697;
   1:  PR[91,3] = PR[90,3] + 29.008;
   1:L PR[91] R[100]mm/sec CNT100;
   1:  PR[91,1] = PR[90,1] + -28.289;
   1:  PR[91,2] = PR[90,2] + -11.407;
   1:  PR[91,3] = PR[90,3] + 29.015;
   1:L PR[91] R[100]mm/sec CNT100;
   1:  PR[91,1] = PR[90,1] + -27.621;
   1:  PR[91,2] = PR[90,2] + -12.094;
   1:  PR[91,3] = PR[90,3] + 29.022;
   1:L PR[91] R[100]mm/sec CNT100;
   1:  PR[91,1] = PR[90,1] + -26.916;
   1:  PR[91,2] = PR[90,2] + -12.748;
   1:  PR[91,3] = PR[90,3] + 29.029;
   1:L PR[91] R[100]mm/sec CNT100;
   1:  PR[91,1] = PR[90,1] + -26.174;
   1:  PR[91,2] = PR[90,2] + -13.367;
   1:  PR[91,3] = PR[90,3] + 29.036;
   1:L PR[91] R[100]mm/sec CNT100;
   1:  PR[91,1] = PR[90,1] + -25.398;
   1:  PR[91,2] = PR[90,2] + -13.952;
   1:  PR[91,3] = PR[90,3] + 29.044;
   1:L PR[91] R[100]mm/sec CNT100;
   1:  PR[91,1] = PR[90,1] + -24.590;
   1:  PR[91,2] = PR[90,2] + -14.499;
   1:  PR[91,3] = PR[90,3] + 29.051;
   1:L PR[91] R[100]mm/sec CNT100;
   1:  PR[91,1] = PR[90,1] + -23.751;
   1:  PR[91,2] = PR[90,2] + -15.008;
   1:  PR[91,3] = PR[90,3] + 29.059;
   1:L PR[91] R[100]mm/sec CNT100;
   1:  PR[91,1] = PR[90,1] + -22.884;
   1:  PR[91,2] = PR[90,2] + -15.477;
   1:  PR[91,3] = PR[90,3] + 29.066;
   1:L PR[91] R[100]mm/sec CNT100;
   1:  PR[91,1] = PR[90,1] + -21.991;
   1:  PR[91,2] = PR[90,2] + -15.905;
   1:  PR[91,3] = PR[90,3] + 29.073;
   1:L PR[91] R[100]mm/sec CNT100;
   1:  PR[91,1] = PR[90,1] + -21.075;
   1:  PR[91,2] = PR[90,2] + -16.289;
   1:  PR[91,3] = PR[90,3] + 29.081;
   1:L PR[91] R[100]mm/sec CNT100;
   1:  PR[91,1] = PR[90,1] + -20.138;
   1:  PR[91,2] = PR[90,2] + -16.629;
   1:  PR[91,3] = PR[90,3] + 29.088;
   1:L PR[91] R[100]mm/sec CNT100;
   1:  PR[91,1] = PR[90,1] + -19.182;
   1:  PR[91,2] = PR[90,2] + -16.922;
   1:  PR[91,3] = PR[90,3] + 29.096;
   1:L PR[91] R[100]mm/sec CNT100;
   1:  PR[91,1] = PR[90,1] + -18.211;
   1:  PR[91,2] = PR[90,2] + -17.168;
   1:  PR[91,3] = PR[90,3] + 29.104;
   1:L PR[91] R[100]mm/sec CNT100;
   1:  PR[91,1] = PR[90,1] + -17.211;
   1:  PR[91,2] = PR[90,2] + -17.368;
   1:  PR[91,3] = PR[90,3] + 29.111;
   1:L PR[91] R[100]mm/sec CNT100;
   1:  PR[91,1] = PR[90,1] + -16.195;
   1:  PR[91,2] = PR[90,2] + -17.522;
   1:  PR[91,3] = PR[90,3] + 29.119;
   1:L PR[91] R[100]mm/sec CNT100;
   1:  PR[91,1] = PR[90,1] + -15.151;
   1:  PR[91,2] = PR[90,2] + -17.626;
   1:  PR[91,3] = PR[90,3] + 29.127;
   1:L PR[91] R[100]mm/sec CNT100;
   1:  PR[91,1] = PR[90,1] + -14.333;
   1:  PR[91,2] = PR[90,2] + -17.670;
   1:  PR[91,3] = PR[90,3] + 29.135;
   1:L PR[91] R[100]mm/sec CNT100;
   1:  PR[91,1] = PR[90,1] + -13.369;
   1:  PR[91,2] = PR[90,2] + -17.680;
   1:  PR[91,3] = PR[90,3] + 29.141;
   1:L PR[91] R[100]mm/sec CNT100;
   1:  PR[91,1] = PR[90,1] + -12.024;
   1:  PR[91,2] = PR[90,2] + -17.616;
   1:  PR[91,3] = PR[90,3] + 29.148;
   1:L PR[91] R[100]mm/sec CNT100;
   1:  PR[91,1] = PR[90,1] + -10.995;
   1:  PR[91,2] = PR[90,2] + -17.507;
   1:  PR[91,3] = PR[90,3] + 29.158;
   1:L PR[91] R[100]mm/sec CNT100;
   1:  PR[91,1] = PR[90,1] + -9.969;
   1:  PR[91,2] = PR[90,2] + -17.345;
   1:  PR[91,3] = PR[90,3] + 29.166;
   1:L PR[91] R[100]mm/sec CNT100;
   1:  PR[91,1] = PR[90,1] + -9.549;
   1:  PR[91,2] = PR[90,2] + -17.262;
   1:  PR[91,3] = PR[90,3] + 29.174;
   1:L PR[91] R[100]mm/sec CNT100;
   1:  PR[91,1] = PR[90,1] + -8.611;
   1:  PR[91,2] = PR[90,2] + -17.045;
   1:  PR[91,3] = PR[90,3] + 29.177;
   1:L PR[91] R[100]mm/sec CNT100;
   1:  PR[91,1] = PR[90,1] + -7.690;
   1:  PR[91,2] = PR[90,2] + -16.783;
   1:  PR[91,3] = PR[90,3] + 29.185;
   1:L PR[91] R[100]mm/sec CNT100;
   1:  PR[91,1] = PR[90,1] + -7.002;
   1:  PR[91,2] = PR[90,2] + -16.556;
   1:  PR[91,3] = PR[90,3] + 29.192;
   1:L PR[91] R[100]mm/sec CNT100;
   1:  PR[91,1] = PR[90,1] + -6.049;
   1:  PR[91,2] = PR[90,2] + -16.194;
   1:  PR[91,3] = PR[90,3] + 29.197;
   1:L PR[91] R[100]mm/sec CNT100;
   1:  PR[91,1] = PR[90,1] + -5.121;
   1:  PR[91,2] = PR[90,2] + -15.785;
   1:  PR[91,3] = PR[90,3] + 29.205;
   1:L PR[91] R[100]mm/sec CNT100;
   1:  PR[91,1] = PR[90,1] + -4.220;
   1:  PR[91,2] = PR[90,2] + -15.332;
   1:  PR[91,3] = PR[90,3] + 29.213;
   1:L PR[91] R[100]mm/sec CNT100;
   1:  PR[91,1] = PR[90,1] + -3.345;
   1:  PR[91,2] = PR[90,2] + -14.834;
   1:  PR[91,3] = PR[90,3] + 29.220;
   1:L PR[91] R[100]mm/sec CNT100;
   1:  PR[91,1] = PR[90,1] + -2.553;
   1:  PR[91,2] = PR[90,2] + -14.330;
   1:  PR[91,3] = PR[90,3] + 29.228;
   1:L PR[91] R[100]mm/sec CNT100;
   1:  PR[91,1] = PR[90,1] + -1.859;
   1:  PR[91,2] = PR[90,2] + -13.840;
   1:  PR[91,3] = PR[90,3] + 29.235;
   1:L PR[91] R[100]mm/sec CNT100;
   1:  PR[91,1] = PR[90,1] + -1.467;
   1:  PR[91,2] = PR[90,2] + -13.594;
   1:  PR[91,3] = PR[90,3] + 29.242;
   1:L PR[91] R[100]mm/sec CNT100;
   1:  PR[91,1] = PR[90,1] + -1.010;
   1:  PR[91,2] = PR[90,2] + -13.406;
   1:  PR[91,3] = PR[90,3] + 29.245;
   1:L PR[91] R[100]mm/sec CNT100;
   1:  PR[91,1] = PR[90,1] + -0.532;
   1:  PR[91,2] = PR[90,2] + -13.297;
   1:  PR[91,3] = PR[90,3] + 29.249;
   1:L PR[91] R[100]mm/sec CNT100;
   1:  PR[91,1] = PR[90,1] + -0.039;
   1:  PR[91,2] = PR[90,2] + -13.266;
   1:  PR[91,3] = PR[90,3] + 29.253;
   1:L PR[91] R[100]mm/sec CNT100;
   1:  PR[91,1] = PR[90,1] + 0.453;
   1:  PR[91,2] = PR[90,2] + -13.325;
   1:  PR[91,3] = PR[90,3] + 29.256;
   1:L PR[91] R[100]mm/sec CNT100;
   1:  PR[91] = PR[90];
   1:  PR[91,1] = PR[90,1] + 1.018;
   1:  PR[91,2] = PR[90,2] + -14.044;
   1:  PR[91,3] = PR[90,3] + 30.590;
   1:L PR[91] R[100]mm/sec CNT100;
   1:  PR[91,1] = PR[90,1] + 1.445;
   1:  PR[91,2] = PR[90,2] + -14.265;
   1:  PR[91,3] = PR[90,3] + 29.264;
   1:L PR[91] R[100]mm/sec CNT100;
   1:  PR[91,1] = PR[90,1] + 2.334;
   1:  PR[91,2] = PR[90,2] + -14.852;
   1:  PR[91,3] = PR[90,3] + 29.267;
   1:L PR[91] R[100]mm/sec CNT100;
   1:  PR[91,1] = PR[90,1] + 3.212;
   1:  PR[91,2] = PR[90,2] + -15.364;
   1:  PR[91,3] = PR[90,3] + 29.276;
   1:L PR[91] R[100]mm/sec CNT100;
   1:  PR[91,1] = PR[90,1] + 4.119;
   1:  PR[91,2] = PR[90,2] + -15.830;
   1:  PR[91,3] = PR[90,3] + 29.283;
   1:L PR[91] R[100]mm/sec CNT100;
   1:  PR[91,1] = PR[90,1] + 5.049;
   1:  PR[91,2] = PR[90,2] + -16.249;
   1:  PR[91,3] = PR[90,3] + 29.291;
   1:L PR[91] R[100]mm/sec CNT100;
   1:  PR[91,1] = PR[90,1] + 6.224;
   1:  PR[91,2] = PR[90,2] + -16.699;
   1:  PR[91,3] = PR[90,3] + 29.299;
   1:L PR[91] R[100]mm/sec CNT100;
   1:  PR[91,1] = PR[90,1] + 7.134;
   1:  PR[91,2] = PR[90,2] + -16.991;
   1:  PR[91,3] = PR[90,3] + 29.309;
   1:L PR[91] R[100]mm/sec CNT100;
   1:  PR[91,1] = PR[90,1] + 8.057;
   1:  PR[91,2] = PR[90,2] + -17.240;
   1:  PR[91,3] = PR[90,3] + 29.316;
   1:L PR[91] R[100]mm/sec CNT100;
   1:  PR[91,1] = PR[90,1] + 8.989;
   1:  PR[91,2] = PR[90,2] + -17.445;
   1:  PR[91,3] = PR[90,3] + 29.323;
   1:L PR[91] R[100]mm/sec CNT100;
   1:  PR[91,1] = PR[90,1] + 9.963;
   1:  PR[91,2] = PR[90,2] + -17.610;
   1:  PR[91,3] = PR[90,3] + 29.331;
   1:L PR[91] R[100]mm/sec CNT100;
   1:  PR[91,1] = PR[90,1] + 10.969;
   1:  PR[91,2] = PR[90,2] + -17.731;
   1:  PR[91,3] = PR[90,3] + 29.338;
   1:L PR[91] R[100]mm/sec CNT100;
   1:  PR[91,1] = PR[90,1] + 11.977;
   1:  PR[91,2] = PR[90,2] + -17.801;
   1:  PR[91,3] = PR[90,3] + 29.346;
   1:L PR[91] R[100]mm/sec CNT100;
   1:  PR[91,1] = PR[90,1] + 12.987;
   1:  PR[91,2] = PR[90,2] + -17.821;
   1:  PR[91,3] = PR[90,3] + 29.354;
   1:L PR[91] R[100]mm/sec CNT100;
   1:  PR[91,1] = PR[90,1] + 13.995;
   1:  PR[91,2] = PR[90,2] + -17.792;
   1:  PR[91,3] = PR[90,3] + 29.361;
